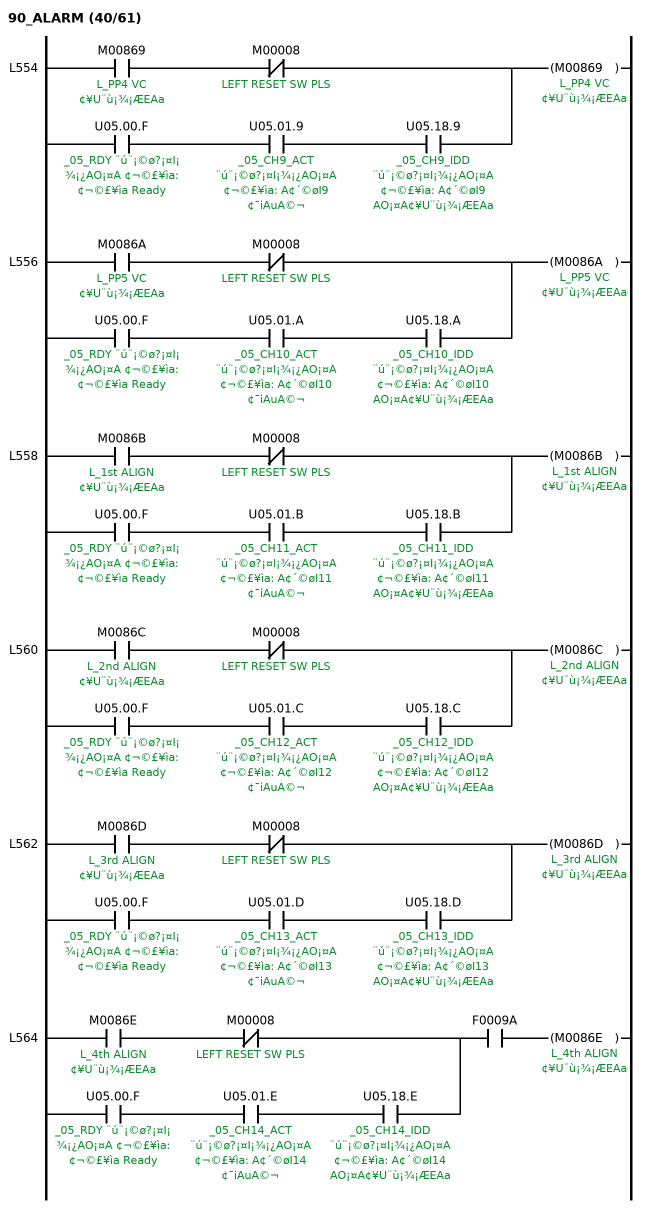
[picture p408: 90_ALARM rungs L554-L564]
; L554
LOAD      M00869	// L_PP4 VC ¢¥U¨ù¡¾¡ÆEAa
AND NOT   M00008	// LEFT RESET SW PLS
LOAD      U05.00.F	// _05_RDY ¨ú¨¡©ø?¡¤I¡¾¡¿AO¡¤A ¢¬©£¥ìa: ¢¬©£¥ìa Ready
AND       U05.01.9	// _05_CH9_ACT ¨ú¨¡©ø?¡¤I¡¾¡¿AO¡¤A ¢¬©£¥ìa: A¢´©øI9 ¢¯iAuA©¬
AND       U05.18.9	// _05_CH9_IDD ¨ú¨¡©ø?¡¤I¡¾¡¿AO¡¤A ¢¬©£¥ìa: A¢´©øI9 AO¡¤A¢¥U¨ù¡¾¡ÆEAa
OR LOAD
OUT       M00869	// L_PP4 VC ¢¥U¨ù¡¾¡ÆEAa
; L556
LOAD      M0086A	// L_PP5 VC ¢¥U¨ù¡¾¡ÆEAa
AND NOT   M00008	// LEFT RESET SW PLS
LOAD      U05.00.F	// _05_RDY ¨ú¨¡©ø?¡¤I¡¾¡¿AO¡¤A ¢¬©£¥ìa: ¢¬©£¥ìa Ready
AND       U05.01.A	// _05_CH10_ACT ¨ú¨¡©ø?¡¤I¡¾¡¿AO¡¤A ¢¬©£¥ìa: A¢´©øI10 ¢¯iAuA©¬
AND       U05.18.A	// _05_CH10_IDD ¨ú¨¡©ø?¡¤I¡¾¡¿AO¡¤A ¢¬©£¥ìa: A¢´©øI10 AO¡¤A¢¥U¨ù¡¾¡ÆEAa
OR LOAD
OUT       M0086A	// L_PP5 VC ¢¥U¨ù¡¾¡ÆEAa
; L558
LOAD      M0086B	// L_1st ALIGN ¢¥U¨ù¡¾¡ÆEAa
AND NOT   M00008	// LEFT RESET SW PLS
LOAD      U05.00.F	// _05_RDY ¨ú¨¡©ø?¡¤I¡¾¡¿AO¡¤A ¢¬©£¥ìa: ¢¬©£¥ìa Ready
AND       U05.01.B	// _05_CH11_ACT ¨ú¨¡©ø?¡¤I¡¾¡¿AO¡¤A ¢¬©£¥ìa: A¢´©øI11 ¢¯iAuA©¬
AND       U05.18.B	// _05_CH11_IDD ¨ú¨¡©ø?¡¤I¡¾¡¿AO¡¤A ¢¬©£¥ìa: A¢´©øI11 AO¡¤A¢¥U¨ù¡¾¡ÆEAa
OR LOAD
OUT       M0086B	// L_1st ALIGN ¢¥U¨ù¡¾¡ÆEAa
; L560
LOAD      M0086C	// L_2nd ALIGN ¢¥U¨ù¡¾¡ÆEAa
AND NOT   M00008	// LEFT RESET SW PLS
LOAD      U05.00.F	// _05_RDY ¨ú¨¡©ø?¡¤I¡¾¡¿AO¡¤A ¢¬©£¥ìa: ¢¬©£¥ìa Ready
AND       U05.01.C	// _05_CH12_ACT ¨ú¨¡©ø?¡¤I¡¾¡¿AO¡¤A ¢¬©£¥ìa: A¢´©øI12 ¢¯iAuA©¬
AND       U05.18.C	// _05_CH12_IDD ¨ú¨¡©ø?¡¤I¡¾¡¿AO¡¤A ¢¬©£¥ìa: A¢´©øI12 AO¡¤A¢¥U¨ù¡¾¡ÆEAa
OR LOAD
OUT       M0086C	// L_2nd ALIGN ¢¥U¨ù¡¾¡ÆEAa
; L562
LOAD      M0086D	// L_3rd ALIGN ¢¥U¨ù¡¾¡ÆEAa
AND NOT   M00008	// LEFT RESET SW PLS
LOAD      U05.00.F	// _05_RDY ¨ú¨¡©ø?¡¤I¡¾¡¿AO¡¤A ¢¬©£¥ìa: ¢¬©£¥ìa Ready
AND       U05.01.D	// _05_CH13_ACT ¨ú¨¡©ø?¡¤I¡¾¡¿AO¡¤A ¢¬©£¥ìa: A¢´©øI13 ¢¯iAuA©¬
AND       U05.18.D	// _05_CH13_IDD ¨ú¨¡©ø?¡¤I¡¾¡¿AO¡¤A ¢¬©£¥ìa: A¢´©øI13 AO¡¤A¢¥U¨ù¡¾¡ÆEAa
OR LOAD
OUT       M0086D	// L_3rd ALIGN ¢¥U¨ù¡¾¡ÆEAa
; L564
LOAD      M0086E	// L_4th ALIGN ¢¥U¨ù¡¾¡ÆEAa
AND NOT   M00008	// LEFT RESET SW PLS
LOAD      U05.00.F	// _05_RDY ¨ú¨¡©ø?¡¤I¡¾¡¿AO¡¤A ¢¬©£¥ìa: ¢¬©£¥ìa Ready
AND       U05.01.E	// _05_CH14_ACT ¨ú¨¡©ø?¡¤I¡¾¡¿AO¡¤A ¢¬©£¥ìa: A¢´©øI14 ¢¯iAuA©¬
AND       U05.18.E	// _05_CH14_IDD ¨ú¨¡©ø?¡¤I¡¾¡¿AO¡¤A ¢¬©£¥ìa: A¢´©øI14 AO¡¤A¢¥U¨ù¡¾¡ÆEAa
OR LOAD
AND       F0009A
OUT       M0086E	// L_4th ALIGN ¢¥U¨ù¡¾¡ÆEAa

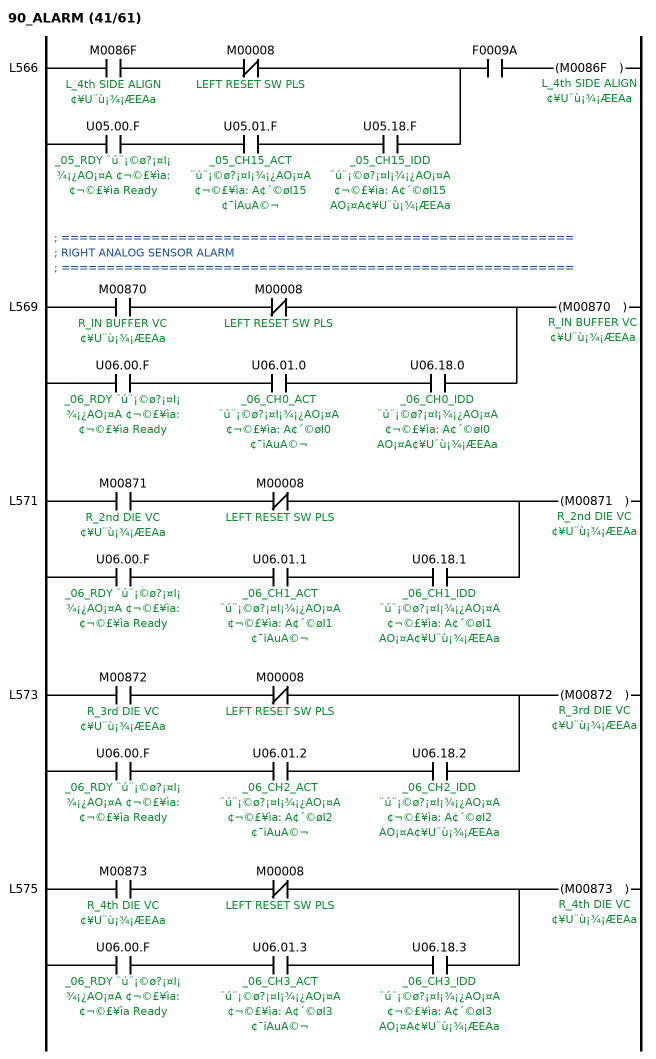
; L566
LOAD      M0086F	// L_4th SIDE ALIGN ¢¥U¨ù¡¾¡ÆEAa
AND NOT   M00008	// LEFT RESET SW PLS
LOAD      U05.00.F	// _05_RDY ¨ú¨¡©ø?¡¤I¡¾¡¿AO¡¤A ¢¬©£¥ìa: ¢¬©£¥ìa Ready
AND       U05.01.F	// _05_CH15_ACT ¨ú¨¡©ø?¡¤I¡¾¡¿AO¡¤A ¢¬©£¥ìa: A¢´©øI15 ¢¯iAuA©¬
AND       U05.18.F	// _05_CH15_IDD ¨ú¨¡©ø?¡¤I¡¾¡¿AO¡¤A ¢¬©£¥ìa: A¢´©øI15 AO¡¤A¢¥U¨ù¡¾¡ÆEAa
OR LOAD
AND       F0009A
OUT       M0086F	// L_4th SIDE ALIGN ¢¥U¨ù¡¾¡ÆEAa
// =========================================================
// 
//        RIGHT ANALOG SENSOR ALARM
// 
// =========================================================
; L569
LOAD      M00870	// R_IN BUFFER VC ¢¥U¨ù¡¾¡ÆEAa
AND NOT   M00008	// LEFT RESET SW PLS
LOAD      U06.00.F	// _06_RDY ¨ú¨¡©ø?¡¤I¡¾¡¿AO¡¤A ¢¬©£¥ìa: ¢¬©£¥ìa Ready
AND       U06.01.0	// _06_CH0_ACT ¨ú¨¡©ø?¡¤I¡¾¡¿AO¡¤A ¢¬©£¥ìa: A¢´©øI0 ¢¯iAuA©¬
AND       U06.18.0	// _06_CH0_IDD ¨ú¨¡©ø?¡¤I¡¾¡¿AO¡¤A ¢¬©£¥ìa: A¢´©øI0 AO¡¤A¢¥U¨ù¡¾¡ÆEAa
OR LOAD
OUT       M00870	// R_IN BUFFER VC ¢¥U¨ù¡¾¡ÆEAa
; L571
LOAD      M00871	// R_2nd DIE VC ¢¥U¨ù¡¾¡ÆEAa
AND NOT   M00008	// LEFT RESET SW PLS
LOAD      U06.00.F	// _06_RDY ¨ú¨¡©ø?¡¤I¡¾¡¿AO¡¤A ¢¬©£¥ìa: ¢¬©£¥ìa Ready
AND       U06.01.1	// _06_CH1_ACT ¨ú¨¡©ø?¡¤I¡¾¡¿AO¡¤A ¢¬©£¥ìa: A¢´©øI1 ¢¯iAuA©¬
AND       U06.18.1	// _06_CH1_IDD ¨ú¨¡©ø?¡¤I¡¾¡¿AO¡¤A ¢¬©£¥ìa: A¢´©øI1 AO¡¤A¢¥U¨ù¡¾¡ÆEAa
OR LOAD
OUT       M00871	// R_2nd DIE VC ¢¥U¨ù¡¾¡ÆEAa
; L573
LOAD      M00872	// R_3rd DIE VC ¢¥U¨ù¡¾¡ÆEAa
AND NOT   M00008	// LEFT RESET SW PLS
LOAD      U06.00.F	// _06_RDY ¨ú¨¡©ø?¡¤I¡¾¡¿AO¡¤A ¢¬©£¥ìa: ¢¬©£¥ìa Ready
AND       U06.01.2	// _06_CH2_ACT ¨ú¨¡©ø?¡¤I¡¾¡¿AO¡¤A ¢¬©£¥ìa: A¢´©øI2 ¢¯iAuA©¬
AND       U06.18.2	// _06_CH2_IDD ¨ú¨¡©ø?¡¤I¡¾¡¿AO¡¤A ¢¬©£¥ìa: A¢´©øI2 AO¡¤A¢¥U¨ù¡¾¡ÆEAa
OR LOAD
OUT       M00872	// R_3rd DIE VC ¢¥U¨ù¡¾¡ÆEAa
; L575
LOAD      M00873	// R_4th DIE VC ¢¥U¨ù¡¾¡ÆEAa
AND NOT   M00008	// LEFT RESET SW PLS
LOAD      U06.00.F	// _06_RDY ¨ú¨¡©ø?¡¤I¡¾¡¿AO¡¤A ¢¬©£¥ìa: ¢¬©£¥ìa Ready
AND       U06.01.3	// _06_CH3_ACT ¨ú¨¡©ø?¡¤I¡¾¡¿AO¡¤A ¢¬©£¥ìa: A¢´©øI3 ¢¯iAuA©¬
AND       U06.18.3	// _06_CH3_IDD ¨ú¨¡©ø?¡¤I¡¾¡¿AO¡¤A ¢¬©£¥ìa: A¢´©øI3 AO¡¤A¢¥U¨ù¡¾¡ÆEAa
OR LOAD
OUT       M00873	// R_4th DIE VC ¢¥U¨ù¡¾¡ÆEAa

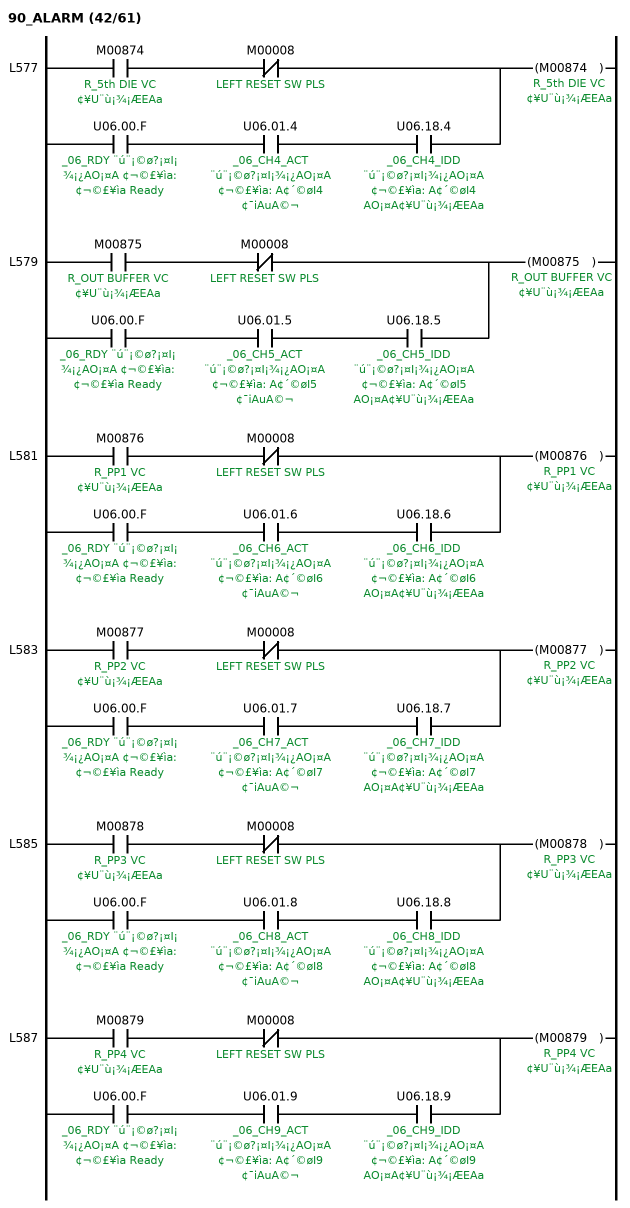
; L577
LOAD      M00874	// R_5th DIE VC ¢¥U¨ù¡¾¡ÆEAa
AND NOT   M00008	// LEFT RESET SW PLS
LOAD      U06.00.F	// _06_RDY ¨ú¨¡©ø?¡¤I¡¾¡¿AO¡¤A ¢¬©£¥ìa: ¢¬©£¥ìa Ready
AND       U06.01.4	// _06_CH4_ACT ¨ú¨¡©ø?¡¤I¡¾¡¿AO¡¤A ¢¬©£¥ìa: A¢´©øI4 ¢¯iAuA©¬
AND       U06.18.4	// _06_CH4_IDD ¨ú¨¡©ø?¡¤I¡¾¡¿AO¡¤A ¢¬©£¥ìa: A¢´©øI4 AO¡¤A¢¥U¨ù¡¾¡ÆEAa
OR LOAD
OUT       M00874	// R_5th DIE VC ¢¥U¨ù¡¾¡ÆEAa
; L579
LOAD      M00875	// R_OUT BUFFER VC ¢¥U¨ù¡¾¡ÆEAa
AND NOT   M00008	// LEFT RESET SW PLS
LOAD      U06.00.F	// _06_RDY ¨ú¨¡©ø?¡¤I¡¾¡¿AO¡¤A ¢¬©£¥ìa: ¢¬©£¥ìa Ready
AND       U06.01.5	// _06_CH5_ACT ¨ú¨¡©ø?¡¤I¡¾¡¿AO¡¤A ¢¬©£¥ìa: A¢´©øI5 ¢¯iAuA©¬
AND       U06.18.5	// _06_CH5_IDD ¨ú¨¡©ø?¡¤I¡¾¡¿AO¡¤A ¢¬©£¥ìa: A¢´©øI5 AO¡¤A¢¥U¨ù¡¾¡ÆEAa
OR LOAD
OUT       M00875	// R_OUT BUFFER VC ¢¥U¨ù¡¾¡ÆEAa
; L581
LOAD      M00876	// R_PP1 VC ¢¥U¨ù¡¾¡ÆEAa
AND NOT   M00008	// LEFT RESET SW PLS
LOAD      U06.00.F	// _06_RDY ¨ú¨¡©ø?¡¤I¡¾¡¿AO¡¤A ¢¬©£¥ìa: ¢¬©£¥ìa Ready
AND       U06.01.6	// _06_CH6_ACT ¨ú¨¡©ø?¡¤I¡¾¡¿AO¡¤A ¢¬©£¥ìa: A¢´©øI6 ¢¯iAuA©¬
AND       U06.18.6	// _06_CH6_IDD ¨ú¨¡©ø?¡¤I¡¾¡¿AO¡¤A ¢¬©£¥ìa: A¢´©øI6 AO¡¤A¢¥U¨ù¡¾¡ÆEAa
OR LOAD
OUT       M00876	// R_PP1 VC ¢¥U¨ù¡¾¡ÆEAa
; L583
LOAD      M00877	// R_PP2 VC ¢¥U¨ù¡¾¡ÆEAa
AND NOT   M00008	// LEFT RESET SW PLS
LOAD      U06.00.F	// _06_RDY ¨ú¨¡©ø?¡¤I¡¾¡¿AO¡¤A ¢¬©£¥ìa: ¢¬©£¥ìa Ready
AND       U06.01.7	// _06_CH7_ACT ¨ú¨¡©ø?¡¤I¡¾¡¿AO¡¤A ¢¬©£¥ìa: A¢´©øI7 ¢¯iAuA©¬
AND       U06.18.7	// _06_CH7_IDD ¨ú¨¡©ø?¡¤I¡¾¡¿AO¡¤A ¢¬©£¥ìa: A¢´©øI7 AO¡¤A¢¥U¨ù¡¾¡ÆEAa
OR LOAD
OUT       M00877	// R_PP2 VC ¢¥U¨ù¡¾¡ÆEAa
; L585
LOAD      M00878	// R_PP3 VC ¢¥U¨ù¡¾¡ÆEAa
AND NOT   M00008	// LEFT RESET SW PLS
LOAD      U06.00.F	// _06_RDY ¨ú¨¡©ø?¡¤I¡¾¡¿AO¡¤A ¢¬©£¥ìa: ¢¬©£¥ìa Ready
AND       U06.01.8	// _06_CH8_ACT ¨ú¨¡©ø?¡¤I¡¾¡¿AO¡¤A ¢¬©£¥ìa: A¢´©øI8 ¢¯iAuA©¬
AND       U06.18.8	// _06_CH8_IDD ¨ú¨¡©ø?¡¤I¡¾¡¿AO¡¤A ¢¬©£¥ìa: A¢´©øI8 AO¡¤A¢¥U¨ù¡¾¡ÆEAa
OR LOAD
OUT       M00878	// R_PP3 VC ¢¥U¨ù¡¾¡ÆEAa
; L587
LOAD      M00879	// R_PP4 VC ¢¥U¨ù¡¾¡ÆEAa
AND NOT   M00008	// LEFT RESET SW PLS
LOAD      U06.00.F	// _06_RDY ¨ú¨¡©ø?¡¤I¡¾¡¿AO¡¤A ¢¬©£¥ìa: ¢¬©£¥ìa Ready
AND       U06.01.9	// _06_CH9_ACT ¨ú¨¡©ø?¡¤I¡¾¡¿AO¡¤A ¢¬©£¥ìa: A¢´©øI9 ¢¯iAuA©¬
AND       U06.18.9	// _06_CH9_IDD ¨ú¨¡©ø?¡¤I¡¾¡¿AO¡¤A ¢¬©£¥ìa: A¢´©øI9 AO¡¤A¢¥U¨ù¡¾¡ÆEAa
OR LOAD
OUT       M00879	// R_PP4 VC ¢¥U¨ù¡¾¡ÆEAa

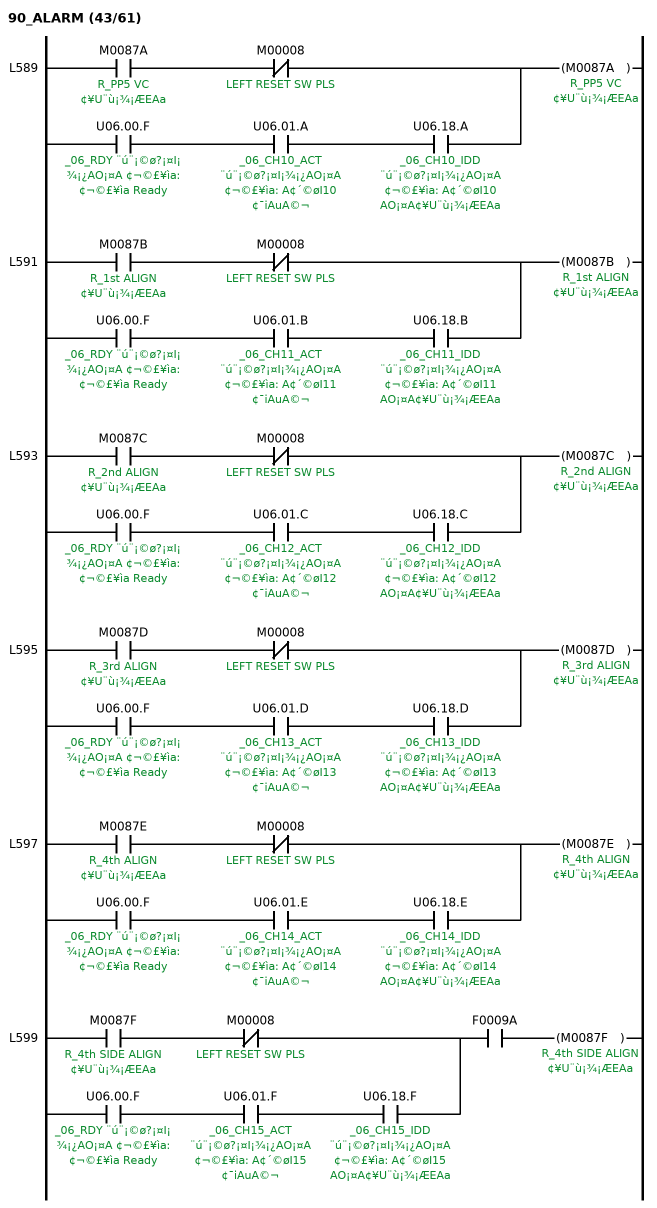
; L589
LOAD      M0087A	// R_PP5 VC ¢¥U¨ù¡¾¡ÆEAa
AND NOT   M00008	// LEFT RESET SW PLS
LOAD      U06.00.F	// _06_RDY ¨ú¨¡©ø?¡¤I¡¾¡¿AO¡¤A ¢¬©£¥ìa: ¢¬©£¥ìa Ready
AND       U06.01.A	// _06_CH10_ACT ¨ú¨¡©ø?¡¤I¡¾¡¿AO¡¤A ¢¬©£¥ìa: A¢´©øI10 ¢¯iAuA©¬
AND       U06.18.A	// _06_CH10_IDD ¨ú¨¡©ø?¡¤I¡¾¡¿AO¡¤A ¢¬©£¥ìa: A¢´©øI10 AO¡¤A¢¥U¨ù¡¾¡ÆEAa
OR LOAD
OUT       M0087A	// R_PP5 VC ¢¥U¨ù¡¾¡ÆEAa
; L591
LOAD      M0087B	// R_1st ALIGN ¢¥U¨ù¡¾¡ÆEAa
AND NOT   M00008	// LEFT RESET SW PLS
LOAD      U06.00.F	// _06_RDY ¨ú¨¡©ø?¡¤I¡¾¡¿AO¡¤A ¢¬©£¥ìa: ¢¬©£¥ìa Ready
AND       U06.01.B	// _06_CH11_ACT ¨ú¨¡©ø?¡¤I¡¾¡¿AO¡¤A ¢¬©£¥ìa: A¢´©øI11 ¢¯iAuA©¬
AND       U06.18.B	// _06_CH11_IDD ¨ú¨¡©ø?¡¤I¡¾¡¿AO¡¤A ¢¬©£¥ìa: A¢´©øI11 AO¡¤A¢¥U¨ù¡¾¡ÆEAa
OR LOAD
OUT       M0087B	// R_1st ALIGN ¢¥U¨ù¡¾¡ÆEAa
; L593
LOAD      M0087C	// R_2nd ALIGN ¢¥U¨ù¡¾¡ÆEAa
AND NOT   M00008	// LEFT RESET SW PLS
LOAD      U06.00.F	// _06_RDY ¨ú¨¡©ø?¡¤I¡¾¡¿AO¡¤A ¢¬©£¥ìa: ¢¬©£¥ìa Ready
AND       U06.01.C	// _06_CH12_ACT ¨ú¨¡©ø?¡¤I¡¾¡¿AO¡¤A ¢¬©£¥ìa: A¢´©øI12 ¢¯iAuA©¬
AND       U06.18.C	// _06_CH12_IDD ¨ú¨¡©ø?¡¤I¡¾¡¿AO¡¤A ¢¬©£¥ìa: A¢´©øI12 AO¡¤A¢¥U¨ù¡¾¡ÆEAa
OR LOAD
OUT       M0087C	// R_2nd ALIGN ¢¥U¨ù¡¾¡ÆEAa
; L595
LOAD      M0087D	// R_3rd ALIGN ¢¥U¨ù¡¾¡ÆEAa
AND NOT   M00008	// LEFT RESET SW PLS
LOAD      U06.00.F	// _06_RDY ¨ú¨¡©ø?¡¤I¡¾¡¿AO¡¤A ¢¬©£¥ìa: ¢¬©£¥ìa Ready
AND       U06.01.D	// _06_CH13_ACT ¨ú¨¡©ø?¡¤I¡¾¡¿AO¡¤A ¢¬©£¥ìa: A¢´©øI13 ¢¯iAuA©¬
AND       U06.18.D	// _06_CH13_IDD ¨ú¨¡©ø?¡¤I¡¾¡¿AO¡¤A ¢¬©£¥ìa: A¢´©øI13 AO¡¤A¢¥U¨ù¡¾¡ÆEAa
OR LOAD
OUT       M0087D	// R_3rd ALIGN ¢¥U¨ù¡¾¡ÆEAa
; L597
LOAD      M0087E	// R_4th ALIGN ¢¥U¨ù¡¾¡ÆEAa
AND NOT   M00008	// LEFT RESET SW PLS
LOAD      U06.00.F	// _06_RDY ¨ú¨¡©ø?¡¤I¡¾¡¿AO¡¤A ¢¬©£¥ìa: ¢¬©£¥ìa Ready
AND       U06.01.E	// _06_CH14_ACT ¨ú¨¡©ø?¡¤I¡¾¡¿AO¡¤A ¢¬©£¥ìa: A¢´©øI14 ¢¯iAuA©¬
AND       U06.18.E	// _06_CH14_IDD ¨ú¨¡©ø?¡¤I¡¾¡¿AO¡¤A ¢¬©£¥ìa: A¢´©øI14 AO¡¤A¢¥U¨ù¡¾¡ÆEAa
OR LOAD
OUT       M0087E	// R_4th ALIGN ¢¥U¨ù¡¾¡ÆEAa
; L599
LOAD      M0087F	// R_4th SIDE ALIGN ¢¥U¨ù¡¾¡ÆEAa
AND NOT   M00008	// LEFT RESET SW PLS
LOAD      U06.00.F	// _06_RDY ¨ú¨¡©ø?¡¤I¡¾¡¿AO¡¤A ¢¬©£¥ìa: ¢¬©£¥ìa Ready
AND       U06.01.F	// _06_CH15_ACT ¨ú¨¡©ø?¡¤I¡¾¡¿AO¡¤A ¢¬©£¥ìa: A¢´©øI15 ¢¯iAuA©¬
AND       U06.18.F	// _06_CH15_IDD ¨ú¨¡©ø?¡¤I¡¾¡¿AO¡¤A ¢¬©£¥ìa: A¢´©øI15 AO¡¤A¢¥U¨ù¡¾¡ÆEAa
OR LOAD
AND       F0009A
OUT       M0087F	// R_4th SIDE ALIGN ¢¥U¨ù¡¾¡ÆEAa

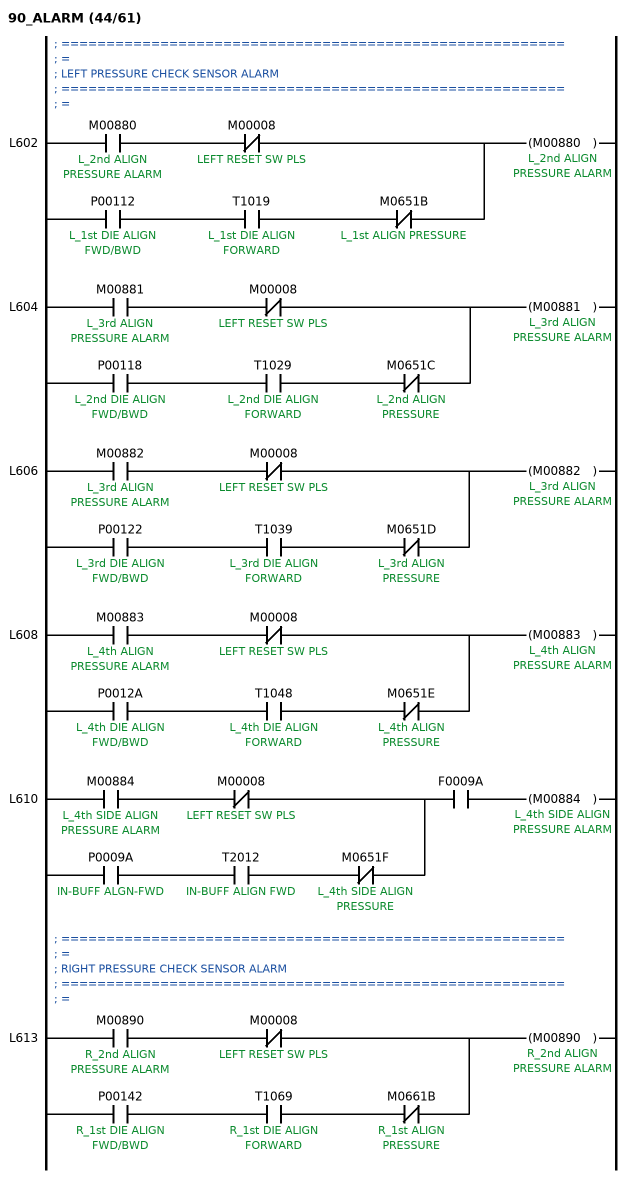
// =========================================================
// 
//        LEFT PRESSURE CHECK SENSOR ALARM
// 
// =========================================================
; L602
LOAD      M00880	// L_2nd ALIGN PRESSURE ALARM
AND NOT   M00008	// LEFT RESET SW PLS
LOAD      P00112	// L_1st DIE ALIGN FWD/BWD
AND       T1019	// L_1st DIE ALIGN FORWARD
AND NOT   M0651B	// L_1st ALIGN PRESSURE
OR LOAD
OUT       M00880	// L_2nd ALIGN PRESSURE ALARM
; L604
LOAD      M00881	// L_3rd ALIGN PRESSURE ALARM
AND NOT   M00008	// LEFT RESET SW PLS
LOAD      P00118	// L_2nd DIE ALIGN FWD/BWD
AND       T1029	// L_2nd DIE ALIGN FORWARD
AND NOT   M0651C	// L_2nd ALIGN PRESSURE
OR LOAD
OUT       M00881	// L_3rd ALIGN PRESSURE ALARM
; L606
LOAD      M00882	// L_3rd ALIGN PRESSURE ALARM
AND NOT   M00008	// LEFT RESET SW PLS
LOAD      P00122	// L_3rd DIE ALIGN FWD/BWD
AND       T1039	// L_3rd DIE ALIGN FORWARD
AND NOT   M0651D	// L_3rd ALIGN PRESSURE
OR LOAD
OUT       M00882	// L_3rd ALIGN PRESSURE ALARM
; L608
LOAD      M00883	// L_4th ALIGN PRESSURE ALARM
AND NOT   M00008	// LEFT RESET SW PLS
LOAD      P0012A	// L_4th DIE ALIGN FWD/BWD
AND       T1048	// L_4th DIE ALIGN FORWARD
AND NOT   M0651E	// L_4th ALIGN PRESSURE
OR LOAD
OUT       M00883	// L_4th ALIGN PRESSURE ALARM
; L610
LOAD      M00884	// L_4th SIDE ALIGN PRESSURE ALARM
AND NOT   M00008	// LEFT RESET SW PLS
LOAD      P0009A	// IN-BUFF ALGN-FWD
AND       T2012	// IN-BUFF ALIGN FWD
AND NOT   M0651F	// L_4th SIDE ALIGN PRESSURE
OR LOAD
AND       F0009A
OUT       M00884	// L_4th SIDE ALIGN PRESSURE ALARM
// =========================================================
// 
//        RIGHT PRESSURE CHECK SENSOR ALARM
// 
// =========================================================
; L613
LOAD      M00890	// R_2nd ALIGN PRESSURE ALARM
AND NOT   M00008	// LEFT RESET SW PLS
LOAD      P00142	// R_1st DIE ALIGN FWD/BWD
AND       T1069	// R_1st DIE ALIGN FORWARD
AND NOT   M0661B	// R_1st ALIGN PRESSURE
OR LOAD
OUT       M00890	// R_2nd ALIGN PRESSURE ALARM

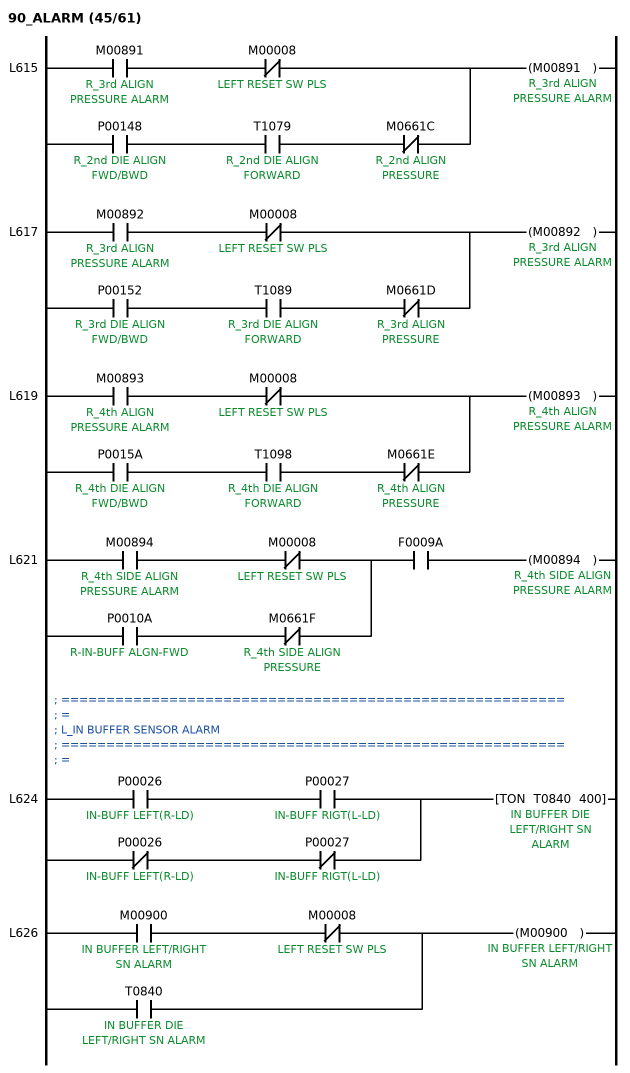
; L615
LOAD      M00891	// R_3rd ALIGN PRESSURE ALARM
AND NOT   M00008	// LEFT RESET SW PLS
LOAD      P00148	// R_2nd DIE ALIGN FWD/BWD
AND       T1079	// R_2nd DIE ALIGN FORWARD
AND NOT   M0661C	// R_2nd ALIGN PRESSURE
OR LOAD
OUT       M00891	// R_3rd ALIGN PRESSURE ALARM
; L617
LOAD      M00892	// R_3rd ALIGN PRESSURE ALARM
AND NOT   M00008	// LEFT RESET SW PLS
LOAD      P00152	// R_3rd DIE ALIGN FWD/BWD
AND       T1089	// R_3rd DIE ALIGN FORWARD
AND NOT   M0661D	// R_3rd ALIGN PRESSURE
OR LOAD
OUT       M00892	// R_3rd ALIGN PRESSURE ALARM
; L619
LOAD      M00893	// R_4th ALIGN PRESSURE ALARM
AND NOT   M00008	// LEFT RESET SW PLS
LOAD      P0015A	// R_4th DIE ALIGN FWD/BWD
AND       T1098	// R_4th DIE ALIGN FORWARD
AND NOT   M0661E	// R_4th ALIGN PRESSURE
OR LOAD
OUT       M00893	// R_4th ALIGN PRESSURE ALARM
; L621
LOAD      M00894	// R_4th SIDE ALIGN PRESSURE ALARM
AND NOT   M00008	// LEFT RESET SW PLS
LOAD      P0010A	// R-IN-BUFF ALGN-FWD
AND NOT   M0661F	// R_4th SIDE ALIGN PRESSURE
OR LOAD
AND       F0009A
OUT       M00894	// R_4th SIDE ALIGN PRESSURE ALARM
// =========================================================
// 
//        L_IN BUFFER SENSOR ALARM
// 
// =========================================================
; L624
LOAD      P00026	// IN-BUFF LEFT(R-LD)
AND       P00027	// IN-BUFF RIGT(L-LD)
LOAD NOT  P00026	// IN-BUFF LEFT(R-LD)
AND NOT   P00027	// IN-BUFF RIGT(L-LD)
OR LOAD
TON       T0840 400	// IN BUFFER DIE LEFT/RIGHT SN ALARM
; L626
LOAD      M00900	// IN BUFFER LEFT/RIGHT SN ALARM
AND NOT   M00008	// LEFT RESET SW PLS
OR        T0840	// IN BUFFER DIE LEFT/RIGHT SN ALARM
OUT       M00900	// IN BUFFER LEFT/RIGHT SN ALARM

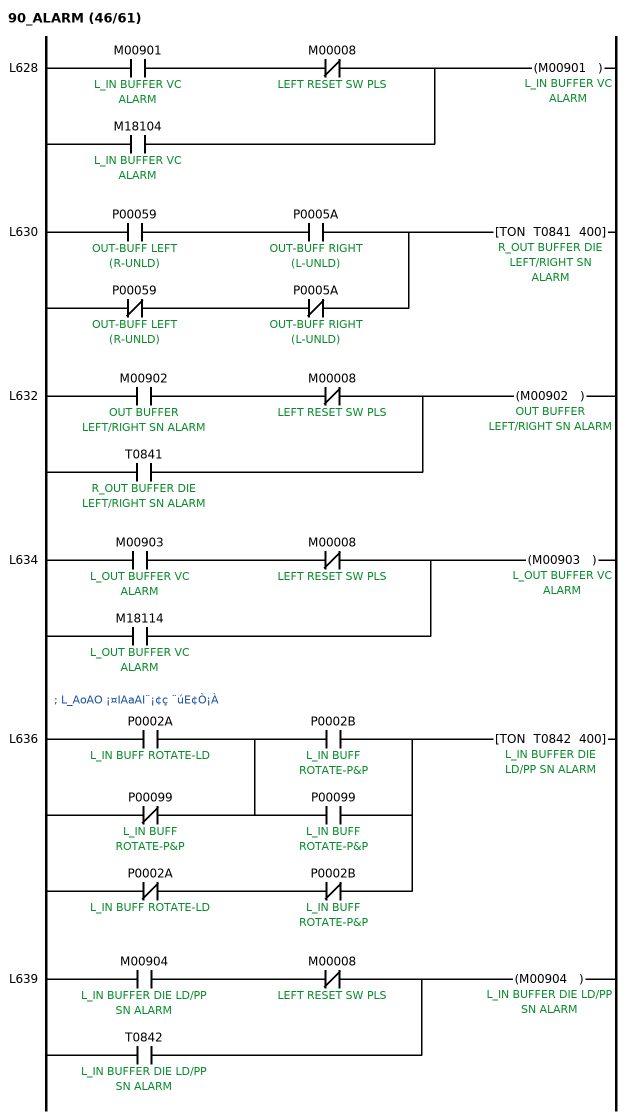
; L628
LOAD      M00901	// L_IN BUFFER VC ALARM
AND NOT   M00008	// LEFT RESET SW PLS
OR        M18104	// L_IN BUFFER VC ALARM
OUT       M00901	// L_IN BUFFER VC ALARM
; L630
LOAD      P00059	// OUT-BUFF LEFT (R-UNLD)
AND       P0005A	// OUT-BUFF RIGHT (L-UNLD)
LOAD NOT  P00059	// OUT-BUFF LEFT (R-UNLD)
AND NOT   P0005A	// OUT-BUFF RIGHT (L-UNLD)
OR LOAD
TON       T0841 400	// R_OUT BUFFER DIE LEFT/RIGHT SN ALARM
; L632
LOAD      M00902	// OUT BUFFER LEFT/RIGHT SN ALARM
AND NOT   M00008	// LEFT RESET SW PLS
OR        T0841	// R_OUT BUFFER DIE LEFT/RIGHT SN ALARM
OUT       M00902	// OUT BUFFER LEFT/RIGHT SN ALARM
; L634
LOAD      M00903	// L_OUT BUFFER VC ALARM
AND NOT   M00008	// LEFT RESET SW PLS
OR        M18114	// L_OUT BUFFER VC ALARM
OUT       M00903	// L_OUT BUFFER VC ALARM
; L636
LOAD      P0002A	// L_IN BUFF ROTATE-LD
OR NOT    P00099	// L_IN BUFF ROTATE-P&P
LOAD      P0002B	// L_IN BUFF ROTATE-P&P
OR        P00099	// L_IN BUFF ROTATE-P&P
AND LOAD
LOAD NOT  P0002A	// L_IN BUFF ROTATE-LD
AND NOT   P0002B	// L_IN BUFF ROTATE-P&P
OR LOAD
TON       T0842 400	// L_IN BUFFER DIE LD/PP SN ALARM
// output comment: L_AoAO ¡¤IAaAI¨¡¢ç ¨úE¢Ò¡À
; L639
LOAD      M00904	// L_IN BUFFER DIE LD/PP SN ALARM
AND NOT   M00008	// LEFT RESET SW PLS
OR        T0842	// L_IN BUFFER DIE LD/PP SN ALARM
OUT       M00904	// L_IN BUFFER DIE LD/PP SN ALARM

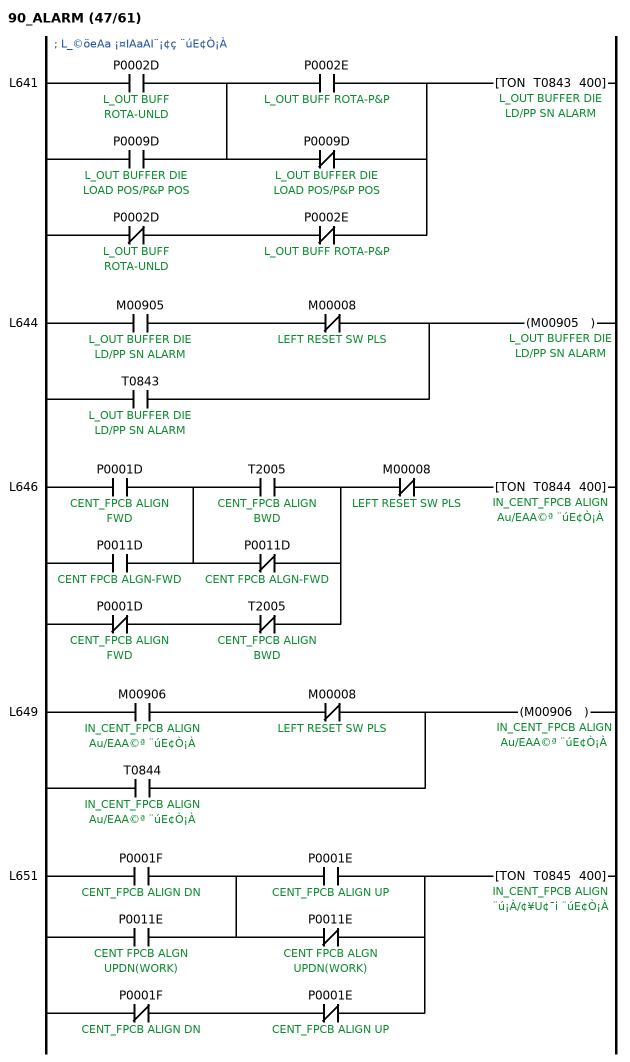
; L641
LOAD      P0002D	// L_OUT BUFF ROTA-UNLD
OR        P0009D	// L_OUT BUFFER DIE LOAD POS/P&P POS
LOAD      P0002E	// L_OUT BUFF ROTA-P&P
OR NOT    P0009D	// L_OUT BUFFER DIE LOAD POS/P&P POS
AND LOAD
LOAD NOT  P0002D	// L_OUT BUFF ROTA-UNLD
AND NOT   P0002E	// L_OUT BUFF ROTA-P&P
OR LOAD
TON       T0843 400	// L_OUT BUFFER DIE LD/PP SN ALARM
// output comment: L_©öeAa ¡¤IAaAI¨¡¢ç ¨úE¢Ò¡À
; L644
LOAD      M00905	// L_OUT BUFFER DIE LD/PP SN ALARM
AND NOT   M00008	// LEFT RESET SW PLS
OR        T0843	// L_OUT BUFFER DIE LD/PP SN ALARM
OUT       M00905	// L_OUT BUFFER DIE LD/PP SN ALARM
; L646
LOAD      P0001D	// CENT_FPCB ALIGN FWD
OR        P0011D	// CENT FPCB ALGN-FWD
LOAD      T2005	// CENT_FPCB ALIGN BWD
OR NOT    P0011D	// CENT FPCB ALGN-FWD
AND LOAD
LOAD NOT  P0001D	// CENT_FPCB ALIGN FWD
AND NOT   T2005	// CENT_FPCB ALIGN BWD
OR LOAD
AND NOT   M00008	// LEFT RESET SW PLS
TON       T0844 400	// IN_CENT_FPCB ALIGN Au/EAA©ª ¨úE¢Ò¡À
; L649
LOAD      M00906	// IN_CENT_FPCB ALIGN Au/EAA©ª ¨úE¢Ò¡À
AND NOT   M00008	// LEFT RESET SW PLS
OR        T0844	// IN_CENT_FPCB ALIGN Au/EAA©ª ¨úE¢Ò¡À
OUT       M00906	// IN_CENT_FPCB ALIGN Au/EAA©ª ¨úE¢Ò¡À
; L651
LOAD      P0001F	// CENT_FPCB ALIGN DN
OR        P0011E	// CENT FPCB ALGN UPDN(WORK)
LOAD      P0001E	// CENT_FPCB ALIGN UP
OR NOT    P0011E	// CENT FPCB ALGN UPDN(WORK)
AND LOAD
LOAD NOT  P0001F	// CENT_FPCB ALIGN DN
AND NOT   P0001E	// CENT_FPCB ALIGN UP
OR LOAD
TON       T0845 400	// IN_CENT_FPCB ALIGN ¨ú¡À/¢¥U¢¯i ¨úE¢Ò¡À

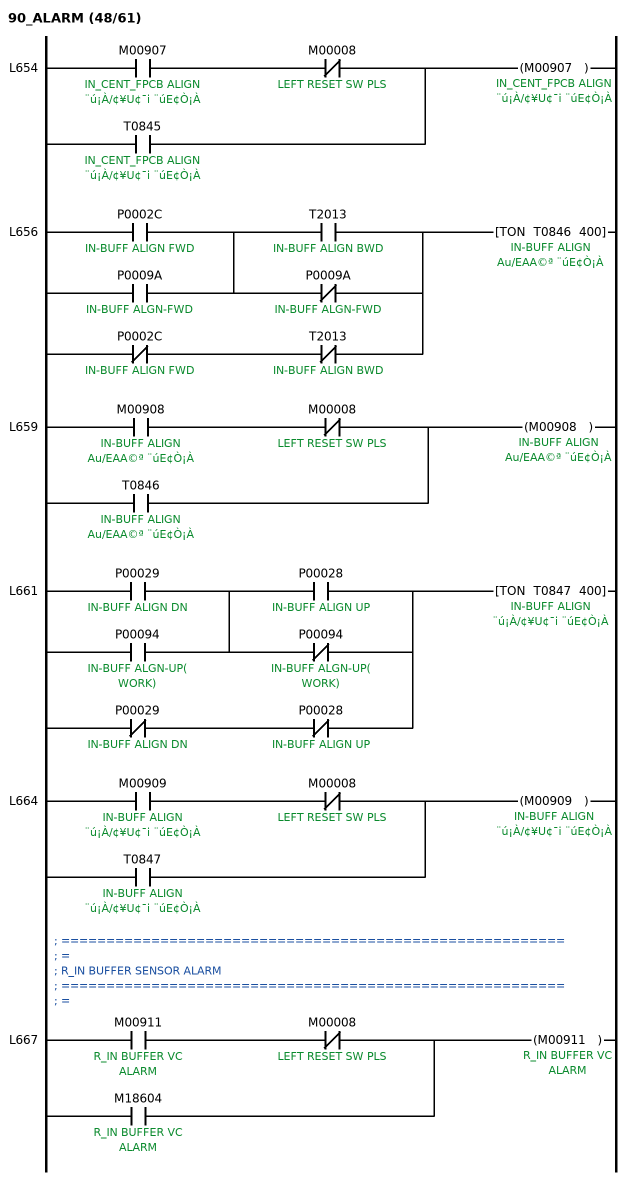
; L654
LOAD      M00907	// IN_CENT_FPCB ALIGN ¨ú¡À/¢¥U¢¯i ¨úE¢Ò¡À
AND NOT   M00008	// LEFT RESET SW PLS
OR        T0845	// IN_CENT_FPCB ALIGN ¨ú¡À/¢¥U¢¯i ¨úE¢Ò¡À
OUT       M00907	// IN_CENT_FPCB ALIGN ¨ú¡À/¢¥U¢¯i ¨úE¢Ò¡À
; L656
LOAD      P0002C	// IN-BUFF ALIGN FWD
OR        P0009A	// IN-BUFF ALGN-FWD
LOAD      T2013	// IN-BUFF ALIGN BWD
OR NOT    P0009A	// IN-BUFF ALGN-FWD
AND LOAD
LOAD NOT  P0002C	// IN-BUFF ALIGN FWD
AND NOT   T2013	// IN-BUFF ALIGN BWD
OR LOAD
TON       T0846 400	// IN-BUFF ALIGN Au/EAA©ª ¨úE¢Ò¡À
; L659
LOAD      M00908	// IN-BUFF ALIGN Au/EAA©ª ¨úE¢Ò¡À
AND NOT   M00008	// LEFT RESET SW PLS
OR        T0846	// IN-BUFF ALIGN Au/EAA©ª ¨úE¢Ò¡À
OUT       M00908	// IN-BUFF ALIGN Au/EAA©ª ¨úE¢Ò¡À
; L661
LOAD      P00029	// IN-BUFF ALIGN DN
OR        P00094	// IN-BUFF ALGN-UP(WORK)
LOAD      P00028	// IN-BUFF ALIGN UP
OR NOT    P00094	// IN-BUFF ALGN-UP(WORK)
AND LOAD
LOAD NOT  P00029	// IN-BUFF ALIGN DN
AND NOT   P00028	// IN-BUFF ALIGN UP
OR LOAD
TON       T0847 400	// IN-BUFF ALIGN ¨ú¡À/¢¥U¢¯i ¨úE¢Ò¡À
; L664
LOAD      M00909	// IN-BUFF ALIGN ¨ú¡À/¢¥U¢¯i ¨úE¢Ò¡À
AND NOT   M00008	// LEFT RESET SW PLS
OR        T0847	// IN-BUFF ALIGN ¨ú¡À/¢¥U¢¯i ¨úE¢Ò¡À
OUT       M00909	// IN-BUFF ALIGN ¨ú¡À/¢¥U¢¯i ¨úE¢Ò¡À
// =========================================================
// 
//        R_IN BUFFER SENSOR ALARM
// 
// =========================================================
; L667
LOAD      M00911	// R_IN BUFFER VC ALARM
AND NOT   M00008	// LEFT RESET SW PLS
OR        M18604	// R_IN BUFFER VC ALARM
OUT       M00911	// R_IN BUFFER VC ALARM

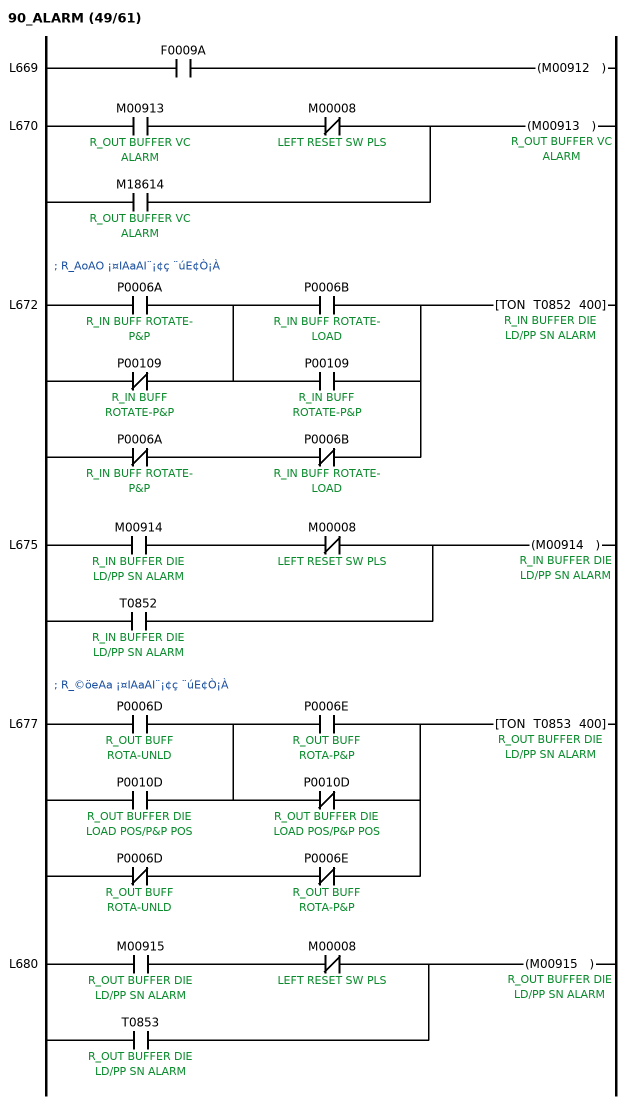
; L669
LOAD      F0009A
OUT       M00912
; L670
LOAD      M00913	// R_OUT BUFFER VC ALARM
AND NOT   M00008	// LEFT RESET SW PLS
OR        M18614	// R_OUT BUFFER VC ALARM
OUT       M00913	// R_OUT BUFFER VC ALARM
; L672
LOAD      P0006A	// R_IN BUFF ROTATE- P&P
OR NOT    P00109	// R_IN BUFF ROTATE-P&P
LOAD      P0006B	// R_IN BUFF ROTATE- LOAD
OR        P00109	// R_IN BUFF ROTATE-P&P
AND LOAD
LOAD NOT  P0006A	// R_IN BUFF ROTATE- P&P
AND NOT   P0006B	// R_IN BUFF ROTATE- LOAD
OR LOAD
TON       T0852 400	// R_IN BUFFER DIE LD/PP SN ALARM
// output comment: R_AoAO ¡¤IAaAI¨¡¢ç ¨úE¢Ò¡À
; L675
LOAD      M00914	// R_IN BUFFER DIE LD/PP SN ALARM
AND NOT   M00008	// LEFT RESET SW PLS
OR        T0852	// R_IN BUFFER DIE LD/PP SN ALARM
OUT       M00914	// R_IN BUFFER DIE LD/PP SN ALARM
; L677
LOAD      P0006D	// R_OUT BUFF ROTA-UNLD
OR        P0010D	// R_OUT BUFFER DIE LOAD POS/P&P POS
LOAD      P0006E	// R_OUT BUFF ROTA-P&P
OR NOT    P0010D	// R_OUT BUFFER DIE LOAD POS/P&P POS
AND LOAD
LOAD NOT  P0006D	// R_OUT BUFF ROTA-UNLD
AND NOT   P0006E	// R_OUT BUFF ROTA-P&P
OR LOAD
TON       T0853 400	// R_OUT BUFFER DIE LD/PP SN ALARM
// output comment: R_©öeAa ¡¤IAaAI¨¡¢ç ¨úE¢Ò¡À
; L680
LOAD      M00915	// R_OUT BUFFER DIE LD/PP SN ALARM
AND NOT   M00008	// LEFT RESET SW PLS
OR        T0853	// R_OUT BUFFER DIE LD/PP SN ALARM
OUT       M00915	// R_OUT BUFFER DIE LD/PP SN ALARM

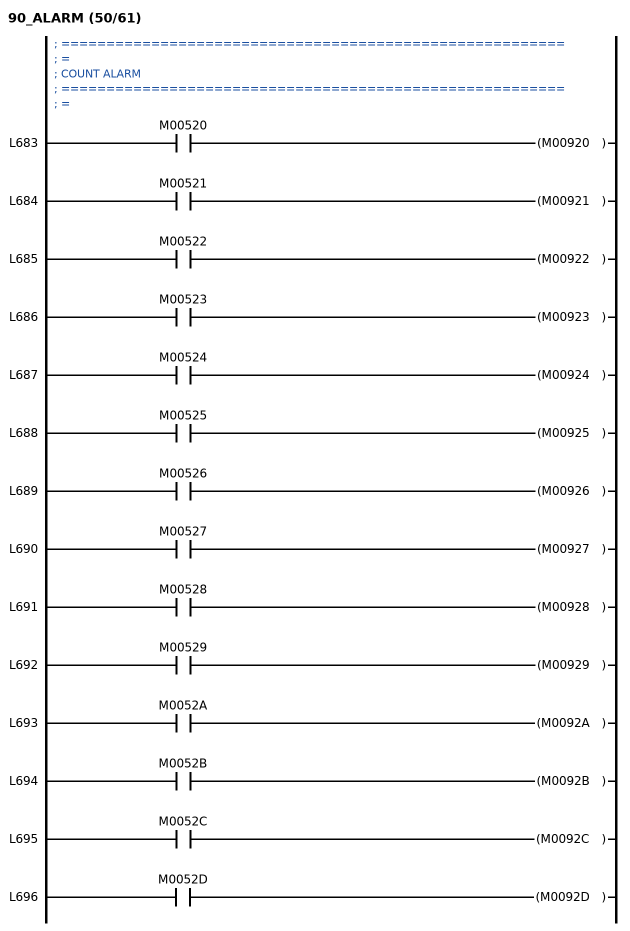
// =========================================================
// 
//       COUNT ALARM
// 
// =========================================================
; L683
LOAD      M00520
OUT       M00920
; L684
LOAD      M00521
OUT       M00921
; L685
LOAD      M00522
OUT       M00922
; L686
LOAD      M00523
OUT       M00923
; L687
LOAD      M00524
OUT       M00924
; L688
LOAD      M00525
OUT       M00925
; L689
LOAD      M00526
OUT       M00926
; L690
LOAD      M00527
OUT       M00927
; L691
LOAD      M00528
OUT       M00928
; L692
LOAD      M00529
OUT       M00929
; L693
LOAD      M0052A
OUT       M0092A
; L694
LOAD      M0052B
OUT       M0092B
; L695
LOAD      M0052C
OUT       M0092C
; L696
LOAD      M0052D
OUT       M0092D

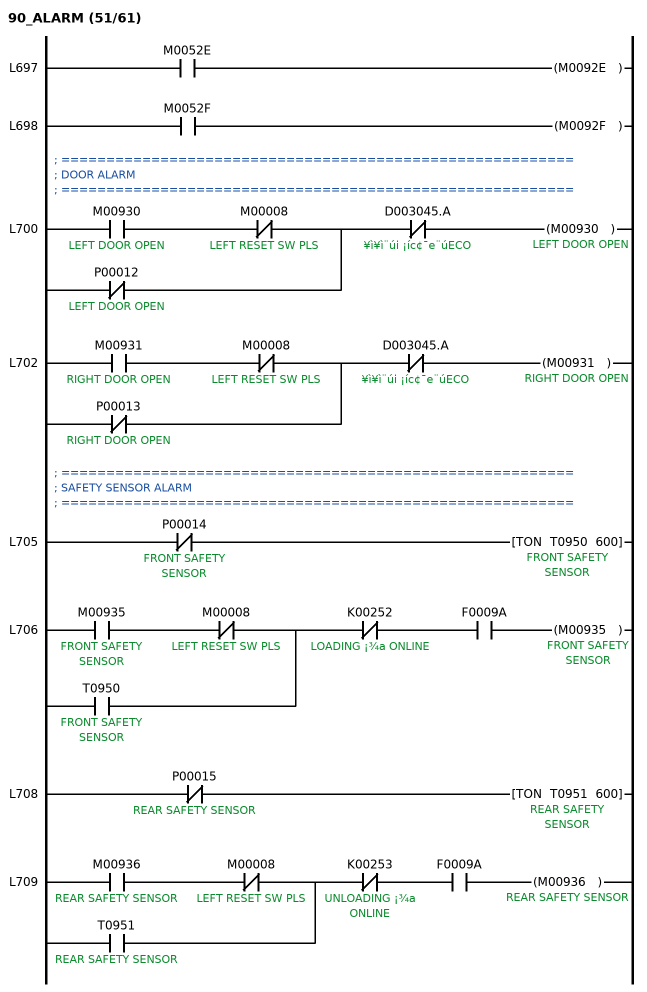
; L697
LOAD      M0052E
OUT       M0092E
; L698
LOAD      M0052F
OUT       M0092F
// =========================================================
// 
//       DOOR ALARM
// 
// =========================================================
; L700
LOAD      M00930	// LEFT DOOR OPEN
AND NOT   M00008	// LEFT RESET SW PLS
OR NOT    P00012	// LEFT DOOR OPEN
AND NOT   D003045.A	// ¥ì¥ì¨úi ¡íc¢¯e¨úECO
OUT       M00930	// LEFT DOOR OPEN
; L702
LOAD      M00931	// RIGHT DOOR OPEN
AND NOT   M00008	// LEFT RESET SW PLS
OR NOT    P00013	// RIGHT DOOR OPEN
AND NOT   D003045.A	// ¥ì¥ì¨úi ¡íc¢¯e¨úECO
OUT       M00931	// RIGHT DOOR OPEN
// =========================================================
// 
//       SAFETY SENSOR ALARM
// 
// =========================================================
; L705
LOAD NOT  P00014	// FRONT SAFETY SENSOR
TON       T0950 600	// FRONT SAFETY SENSOR
; L706
LOAD      M00935	// FRONT SAFETY SENSOR
AND NOT   M00008	// LEFT RESET SW PLS
OR        T0950	// FRONT SAFETY SENSOR
AND NOT   K00252	// LOADING ¡¾a ONLINE
AND       F0009A
OUT       M00935	// FRONT SAFETY SENSOR
; L708
LOAD NOT  P00015	// REAR SAFETY SENSOR
TON       T0951 600	// REAR SAFETY SENSOR
; L709
LOAD      M00936	// REAR SAFETY SENSOR
AND NOT   M00008	// LEFT RESET SW PLS
OR        T0951	// REAR SAFETY SENSOR
AND NOT   K00253	// UNLOADING ¡¾a ONLINE
AND       F0009A
OUT       M00936	// REAR SAFETY SENSOR

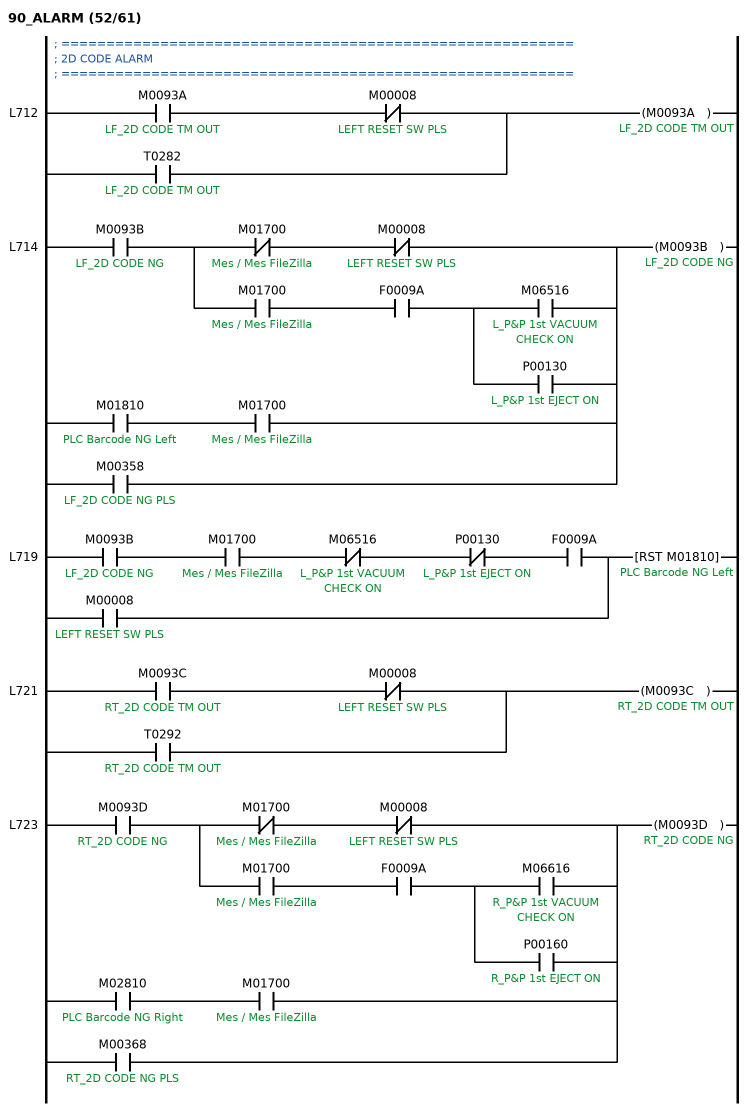
// =========================================================
// 
//       2D CODE ALARM
// 
// =========================================================
; L712
LOAD      M0093A	// LF_2D CODE TM OUT
AND NOT   M00008	// LEFT RESET SW PLS
OR        T0282	// LF_2D CODE TM OUT
OUT       M0093A	// LF_2D CODE TM OUT
; L714
LOAD      M0093B	// LF_2D CODE NG
LOAD NOT  M01700	// Mes / Mes FileZilla
AND NOT   M00008	// LEFT RESET SW PLS
LOAD      M01700	// Mes / Mes FileZilla
AND       F0009A
LOAD      M06516	// L_P&P 1st VACUUM CHECK ON
OR        P00130	// L_P&P 1st EJECT ON
AND LOAD
OR LOAD
AND LOAD
LOAD      M01810	// PLC Barcode NG Left
AND       M01700	// Mes / Mes FileZilla
OR LOAD
OR        M00358	// LF_2D CODE NG PLS
OUT       M0093B	// LF_2D CODE NG
; L719
LOAD      M0093B	// LF_2D CODE NG
AND       M01700	// Mes / Mes FileZilla
AND NOT   M06516	// L_P&P 1st VACUUM CHECK ON
AND NOT   P00130	// L_P&P 1st EJECT ON
AND       F0009A
OR        M00008	// LEFT RESET SW PLS
RST       M01810	// PLC Barcode NG Left
; L721
LOAD      M0093C	// RT_2D CODE TM OUT
AND NOT   M00008	// LEFT RESET SW PLS
OR        T0292	// RT_2D CODE TM OUT
OUT       M0093C	// RT_2D CODE TM OUT
; L723
LOAD      M0093D	// RT_2D CODE NG
LOAD NOT  M01700	// Mes / Mes FileZilla
AND NOT   M00008	// LEFT RESET SW PLS
LOAD      M01700	// Mes / Mes FileZilla
AND       F0009A
LOAD      M06616	// R_P&P 1st VACUUM CHECK ON
OR        P00160	// R_P&P 1st EJECT ON
AND LOAD
OR LOAD
AND LOAD
LOAD      M02810	// PLC Barcode NG Right
AND       M01700	// Mes / Mes FileZilla
OR LOAD
OR        M00368	// RT_2D CODE NG PLS
OUT       M0093D	// RT_2D CODE NG

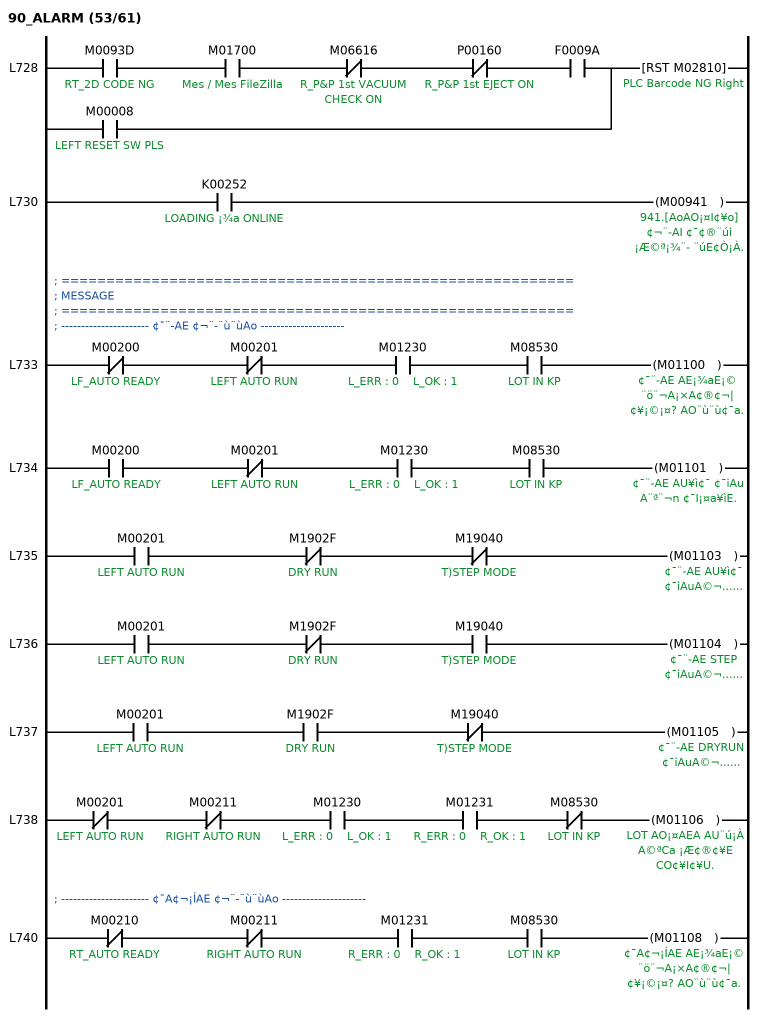
; L728
LOAD      M0093D	// RT_2D CODE NG
AND       M01700	// Mes / Mes FileZilla
AND NOT   M06616	// R_P&P 1st VACUUM CHECK ON
AND NOT   P00160	// R_P&P 1st EJECT ON
AND       F0009A
OR        M00008	// LEFT RESET SW PLS
RST       M02810	// PLC Barcode NG Right
; L730
LOAD      K00252	// LOADING ¡¾a ONLINE
OUT       M00941	// 941.[AoAO¡¤I¢¥o] ¢¬¨­AI ¢¯¢®¨úi ¡Æ©ª¡¾¨­ ¨úE¢Ò¡À.
// =========================================================
// 
//       MESSAGE
// 
// =========================================================
// ---------------------- ¢¯¨­AE ¢¬¨­¨ù¨ùAo ---------------------
; L733
LOAD NOT  M00200	// LF_AUTO READY
AND NOT   M00201	// LEFT AUTO RUN
AND       M01230	// L_ERR : 0    L_OK : 1
AND       M08530	// LOT IN KP
OUT       M01100	// ¢¯¨­AE AE¡¾aE¡© ¨ö¨¬A¡×A¢®¢¬| ¢¥¡©¡¤? AO¨ù¨ù¢¯a.
; L734
LOAD      M00200	// LF_AUTO READY
AND NOT   M00201	// LEFT AUTO RUN
AND       M01230	// L_ERR : 0    L_OK : 1
AND       M08530	// LOT IN KP
OUT       M01101	// ¢¯¨­AE AU¥ì¢¯ ¢¯iAu A¨ª¨¬n ¢¯I¡¤a¥ìE.
; L735
LOAD      M00201	// LEFT AUTO RUN
AND NOT   M1902F	// DRY RUN
AND NOT   M19040	// T)STEP MODE
OUT       M01103	// ¢¯¨­AE AU¥ì¢¯ ¢¯iAuA©¬......
; L736
LOAD      M00201	// LEFT AUTO RUN
AND NOT   M1902F	// DRY RUN
AND       M19040	// T)STEP MODE
OUT       M01104	// ¢¯¨­AE STEP ¢¯iAuA©¬......
; L737
LOAD      M00201	// LEFT AUTO RUN
AND       M1902F	// DRY RUN
AND NOT   M19040	// T)STEP MODE
OUT       M01105	// ¢¯¨­AE DRYRUN ¢¯iAuA©¬......
; L738
LOAD NOT  M00201	// LEFT AUTO RUN
AND NOT   M00211	// RIGHT AUTO RUN
AND       M01230	// L_ERR : 0    L_OK : 1
AND       M01231	// R_ERR : 0    R_OK : 1
AND NOT   M08530	// LOT IN KP
OUT       M01106	// LOT AO¡¤AEA AU¨ú¡À A©ªCa ¡Æ¢®¢¥E CO¢¥I¢¥U.
// ---------------------- ¢¯A¢¬¡ÍAE ¢¬¨­¨ù¨ùAo ---------------------
; L740
LOAD NOT  M00210	// RT_AUTO READY
AND NOT   M00211	// RIGHT AUTO RUN
AND       M01231	// R_ERR : 0    R_OK : 1
AND       M08530	// LOT IN KP
OUT       M01108	// ¢¯A¢¬¡ÍAE AE¡¾aE¡© ¨ö¨¬A¡×A¢®¢¬| ¢¥¡©¡¤? AO¨ù¨ù¢¯a.

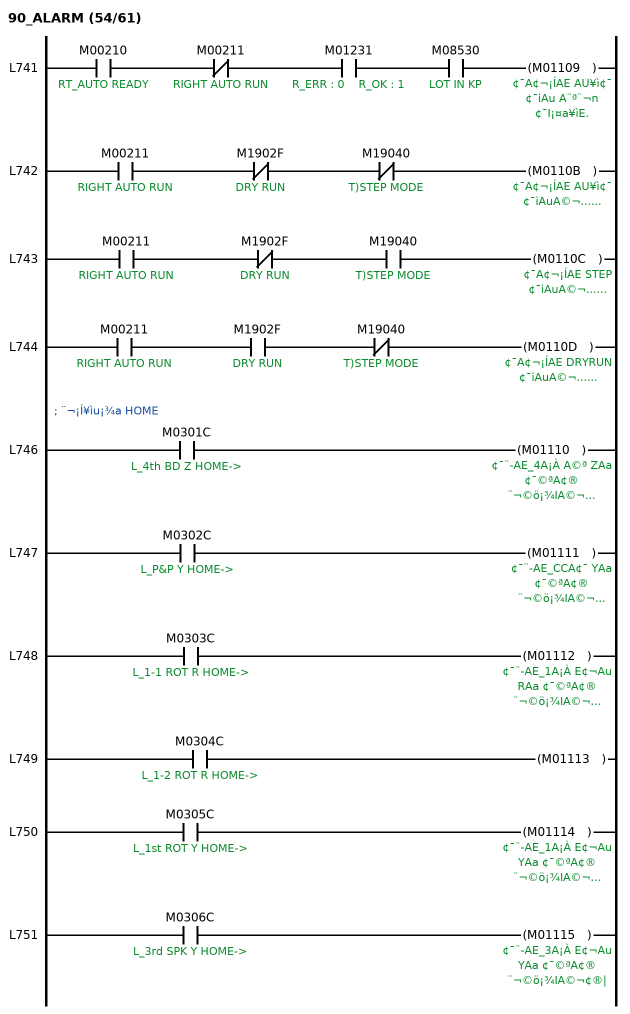
; L741
LOAD      M00210	// RT_AUTO READY
AND NOT   M00211	// RIGHT AUTO RUN
AND       M01231	// R_ERR : 0    R_OK : 1
AND       M08530	// LOT IN KP
OUT       M01109	// ¢¯A¢¬¡ÍAE AU¥ì¢¯ ¢¯iAu A¨ª¨¬n ¢¯I¡¤a¥ìE.
; L742
LOAD      M00211	// RIGHT AUTO RUN
AND NOT   M1902F	// DRY RUN
AND NOT   M19040	// T)STEP MODE
OUT       M0110B	// ¢¯A¢¬¡ÍAE AU¥ì¢¯ ¢¯iAuA©¬......
; L743
LOAD      M00211	// RIGHT AUTO RUN
AND NOT   M1902F	// DRY RUN
AND       M19040	// T)STEP MODE
OUT       M0110C	// ¢¯A¢¬¡ÍAE STEP ¢¯iAuA©¬......
; L744
LOAD      M00211	// RIGHT AUTO RUN
AND       M1902F	// DRY RUN
AND NOT   M19040	// T)STEP MODE
OUT       M0110D	// ¢¯A¢¬¡ÍAE DRYRUN ¢¯iAuA©¬......
// ¨¬¡Í¥ìu¡¾a HOME
; L746
LOAD      M0301C	// L_4th BD Z HOME->
OUT       M01110	// ¢¯¨­AE_4A¡À A©ª ZAa ¢¯©ªA¢® ¨¬©ö¡¾IA©¬...
; L747
LOAD      M0302C	// L_P&P Y HOME->
OUT       M01111	// ¢¯¨­AE_CCA¢¯ YAa ¢¯©ªA¢® ¨¬©ö¡¾IA©¬...
; L748
LOAD      M0303C	// L_1-1 ROT R HOME->
OUT       M01112	// ¢¯¨­AE_1A¡À E¢¬Au RAa ¢¯©ªA¢® ¨¬©ö¡¾IA©¬...
; L749
LOAD      M0304C	// L_1-2 ROT R HOME->
OUT       M01113
; L750
LOAD      M0305C	// L_1st ROT Y HOME->
OUT       M01114	// ¢¯¨­AE_1A¡À E¢¬Au YAa ¢¯©ªA¢® ¨¬©ö¡¾IA©¬...
; L751
LOAD      M0306C	// L_3rd SPK Y HOME->
OUT       M01115	// ¢¯¨­AE_3A¡À E¢¬Au YAa ¢¯©ªA¢® ¨¬©ö¡¾IA©¬¢®|

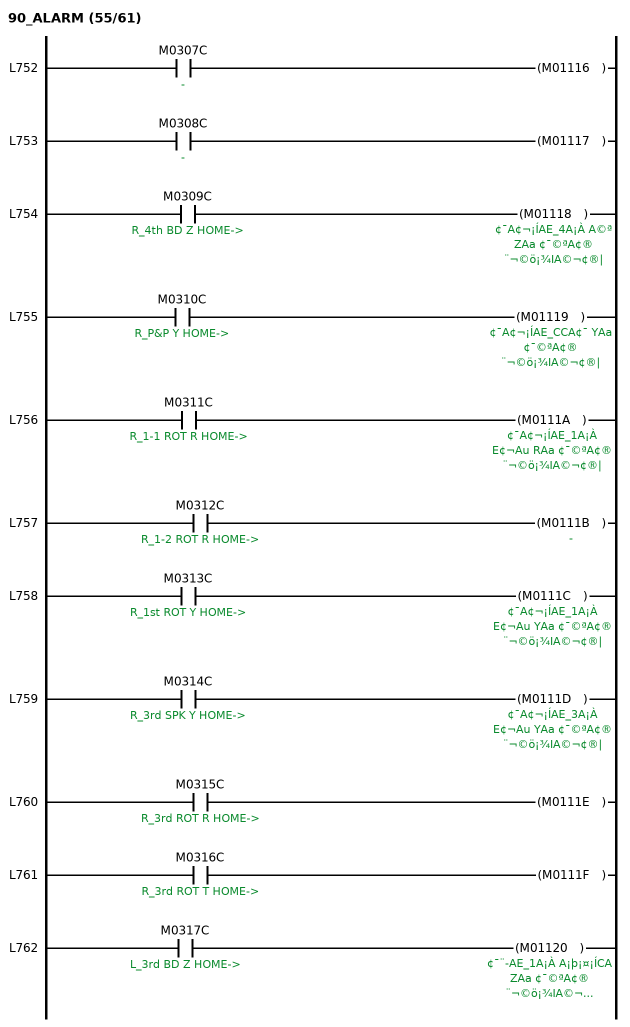
; L752
LOAD      M0307C	// -
OUT       M01116
; L753
LOAD      M0308C	// -
OUT       M01117
; L754
LOAD      M0309C	// R_4th BD Z HOME->
OUT       M01118	// ¢¯A¢¬¡ÍAE_4A¡À A©ª ZAa ¢¯©ªA¢® ¨¬©ö¡¾IA©¬¢®|
; L755
LOAD      M0310C	// R_P&P Y HOME->
OUT       M01119	// ¢¯A¢¬¡ÍAE_CCA¢¯ YAa ¢¯©ªA¢® ¨¬©ö¡¾IA©¬¢®|
; L756
LOAD      M0311C	// R_1-1 ROT R HOME->
OUT       M0111A	// ¢¯A¢¬¡ÍAE_1A¡À E¢¬Au RAa ¢¯©ªA¢® ¨¬©ö¡¾IA©¬¢®|
; L757
LOAD      M0312C	// R_1-2 ROT R HOME->
OUT       M0111B	// -
; L758
LOAD      M0313C	// R_1st ROT Y HOME->
OUT       M0111C	// ¢¯A¢¬¡ÍAE_1A¡À E¢¬Au YAa ¢¯©ªA¢® ¨¬©ö¡¾IA©¬¢®|
; L759
LOAD      M0314C	// R_3rd SPK Y HOME->
OUT       M0111D	// ¢¯A¢¬¡ÍAE_3A¡À E¢¬Au YAa ¢¯©ªA¢® ¨¬©ö¡¾IA©¬¢®|
; L760
LOAD      M0315C	// R_3rd ROT R HOME->
OUT       M0111E
; L761
LOAD      M0316C	// R_3rd ROT T HOME->
OUT       M0111F
; L762
LOAD      M0317C	// L_3rd BD Z HOME->
OUT       M01120	// ¢¯¨­AE_1A¡À A¡þ¡¤¡ÍCA ZAa ¢¯©ªA¢® ¨¬©ö¡¾IA©¬...

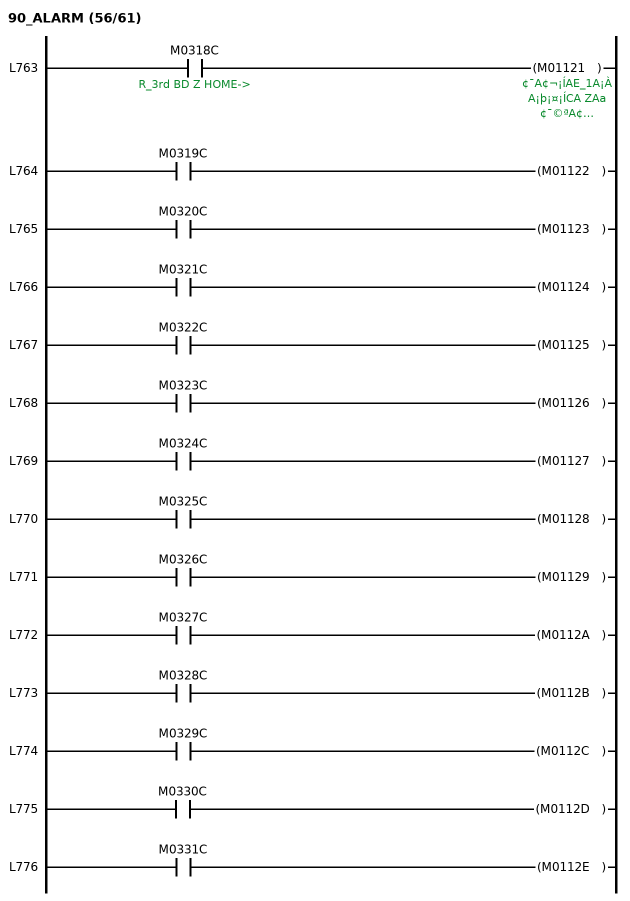
; L763
LOAD      M0318C	// R_3rd BD Z HOME->
OUT       M01121	// ¢¯A¢¬¡ÍAE_1A¡À A¡þ¡¤¡ÍCA ZAa ¢¯©ªA¢® ¨¬©ö¡¾IA©¬...
; L764
LOAD      M0319C
OUT       M01122
; L765
LOAD      M0320C
OUT       M01123
; L766
LOAD      M0321C
OUT       M01124
; L767
LOAD      M0322C
OUT       M01125
; L768
LOAD      M0323C
OUT       M01126
; L769
LOAD      M0324C
OUT       M01127
; L770
LOAD      M0325C
OUT       M01128
; L771
LOAD      M0326C
OUT       M01129
; L772
LOAD      M0327C
OUT       M0112A
; L773
LOAD      M0328C
OUT       M0112B
; L774
LOAD      M0329C
OUT       M0112C
; L775
LOAD      M0330C
OUT       M0112D
; L776
LOAD      M0331C
OUT       M0112E

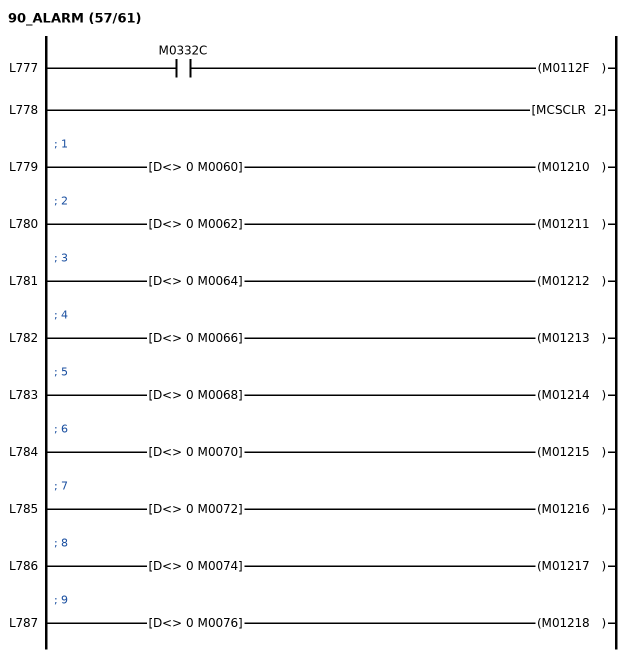
; L777
LOAD      M0332C
OUT       M0112F
; L778
MCSCLR    2
; L779
LOADD<>   0 M0060
OUT       M01210
// output comment: 1
; L780
LOADD<>   0 M0062
OUT       M01211
// output comment: 2
; L781
LOADD<>   0 M0064
OUT       M01212
// output comment: 3
; L782
LOADD<>   0 M0066
OUT       M01213
// output comment: 4
; L783
LOADD<>   0 M0068
OUT       M01214
// output comment: 5
; L784
LOADD<>   0 M0070
OUT       M01215
// output comment: 6
; L785
LOADD<>   0 M0072
OUT       M01216
// output comment: 7
; L786
LOADD<>   0 M0074
OUT       M01217
// output comment: 8
; L787
LOADD<>   0 M0076
OUT       M01218
// output comment: 9

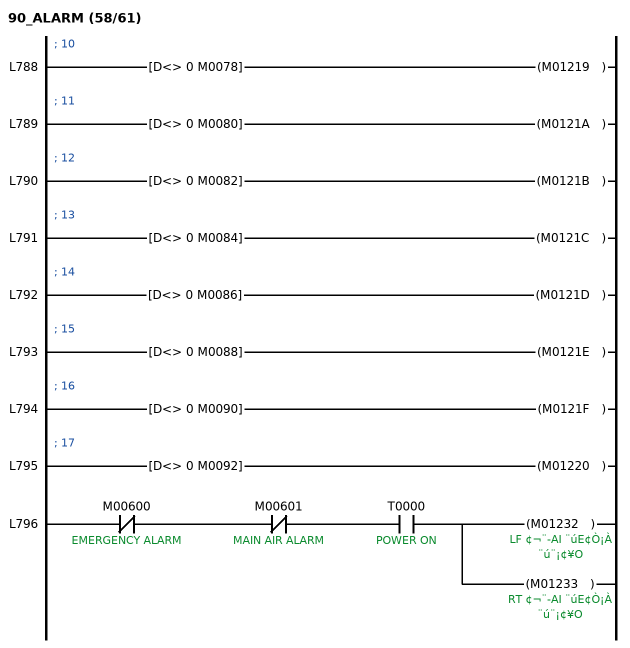
; L788
LOADD<>   0 M0078
OUT       M01219
// output comment: 10
; L789
LOADD<>   0 M0080
OUT       M0121A
// output comment: 11
; L790
LOADD<>   0 M0082
OUT       M0121B
// output comment: 12
; L791
LOADD<>   0 M0084
OUT       M0121C
// output comment: 13
; L792
LOADD<>   0 M0086
OUT       M0121D
// output comment: 14
; L793
LOADD<>   0 M0088
OUT       M0121E
// output comment: 15
; L794
LOADD<>   0 M0090
OUT       M0121F
// output comment: 16
; L795
LOADD<>   0 M0092
OUT       M01220
// output comment: 17
; L796
LOAD NOT  M00600	// EMERGENCY ALARM
AND NOT   M00601	// MAIN AIR ALARM
AND       T0000	// POWER ON
OUT       M01232	// LF ¢¬¨­AI ¨úE¢Ò¡À ¨ú¨¡¢¥O
OUT       M01233	// RT ¢¬¨­AI ¨úE¢Ò¡À ¨ú¨¡¢¥O

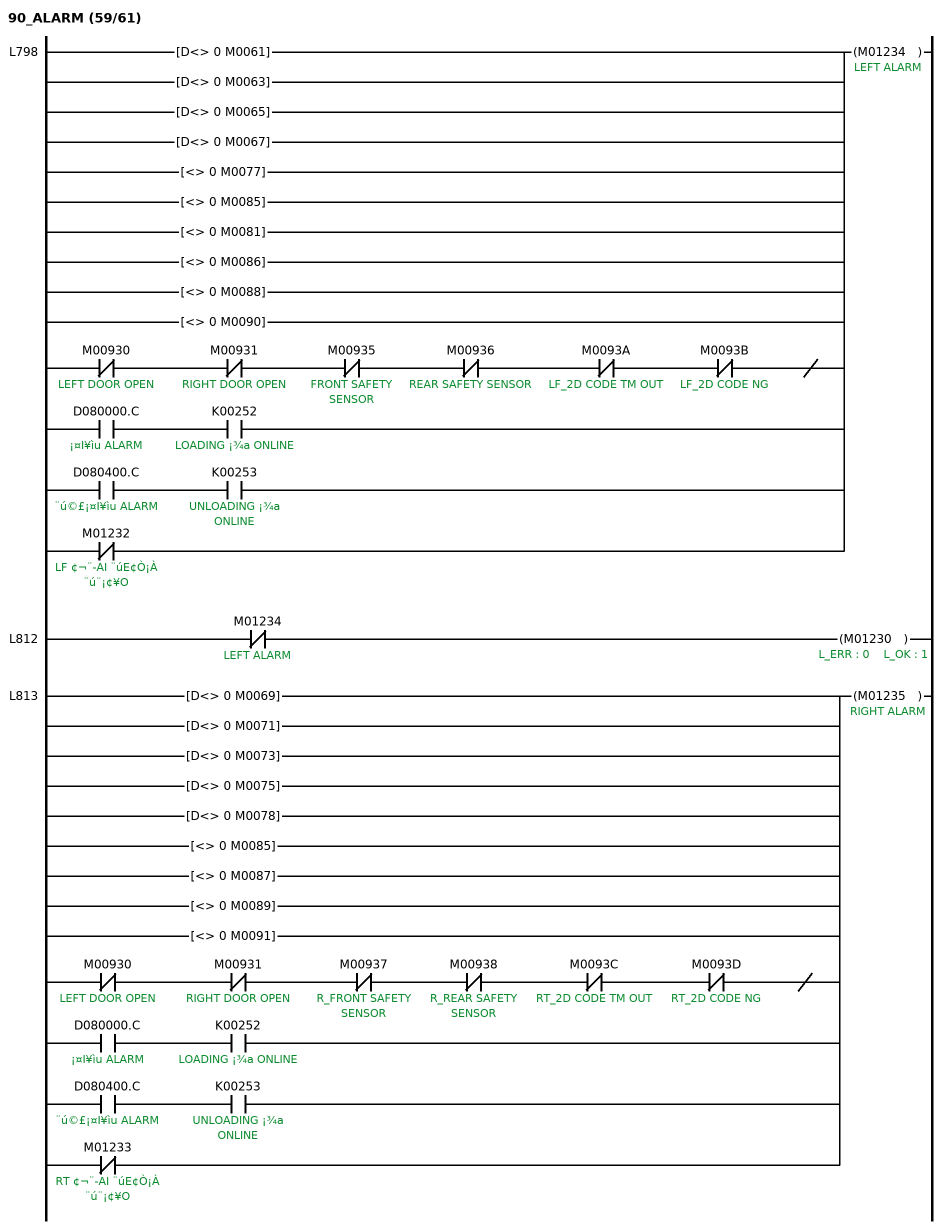
; L798
LOADD<>   0 M0061
ORD<>     0 M0063
ORD<>     0 M0065
ORD<>     0 M0067
OR<>      0 M0077
OR<>      0 M0085
OR<>      0 M0081
OR<>      0 M0086
OR<>      0 M0088
OR<>      0 M0090
LOAD NOT  M00930	// LEFT DOOR OPEN
AND NOT   M00931	// RIGHT DOOR OPEN
AND NOT   M00935	// FRONT SAFETY SENSOR
AND NOT   M00936	// REAR SAFETY SENSOR
AND NOT   M0093A	// LF_2D CODE TM OUT
AND NOT   M0093B	// LF_2D CODE NG
NOT
OR LOAD
LOAD      D080000.C	// ¡¤I¥ìu ALARM
AND       K00252	// LOADING ¡¾a ONLINE
OR LOAD
LOAD      D080400.C	// ¨ú©£¡¤I¥ìu ALARM
AND       K00253	// UNLOADING ¡¾a ONLINE
OR LOAD
OR NOT    M01232	// LF ¢¬¨­AI ¨úE¢Ò¡À ¨ú¨¡¢¥O
OUT       M01234	// LEFT ALARM
; L812
LOAD NOT  M01234	// LEFT ALARM
OUT       M01230	// L_ERR : 0    L_OK : 1
; L813
LOADD<>   0 M0069
ORD<>     0 M0071
ORD<>     0 M0073
ORD<>     0 M0075
ORD<>     0 M0078
OR<>      0 M0085
OR<>      0 M0087
OR<>      0 M0089
OR<>      0 M0091
LOAD NOT  M00930	// LEFT DOOR OPEN
AND NOT   M00931	// RIGHT DOOR OPEN
AND NOT   M00937	// R_FRONT SAFETY SENSOR
AND NOT   M00938	// R_REAR SAFETY SENSOR
AND NOT   M0093C	// RT_2D CODE TM OUT
AND NOT   M0093D	// RT_2D CODE NG
NOT
OR LOAD
LOAD      D080000.C	// ¡¤I¥ìu ALARM
AND       K00252	// LOADING ¡¾a ONLINE
OR LOAD
LOAD      D080400.C	// ¨ú©£¡¤I¥ìu ALARM
AND       K00253	// UNLOADING ¡¾a ONLINE
OR LOAD
OR NOT    M01233	// RT ¢¬¨­AI ¨úE¢Ò¡À ¨ú¨¡¢¥O
OUT       M01235	// RIGHT ALARM

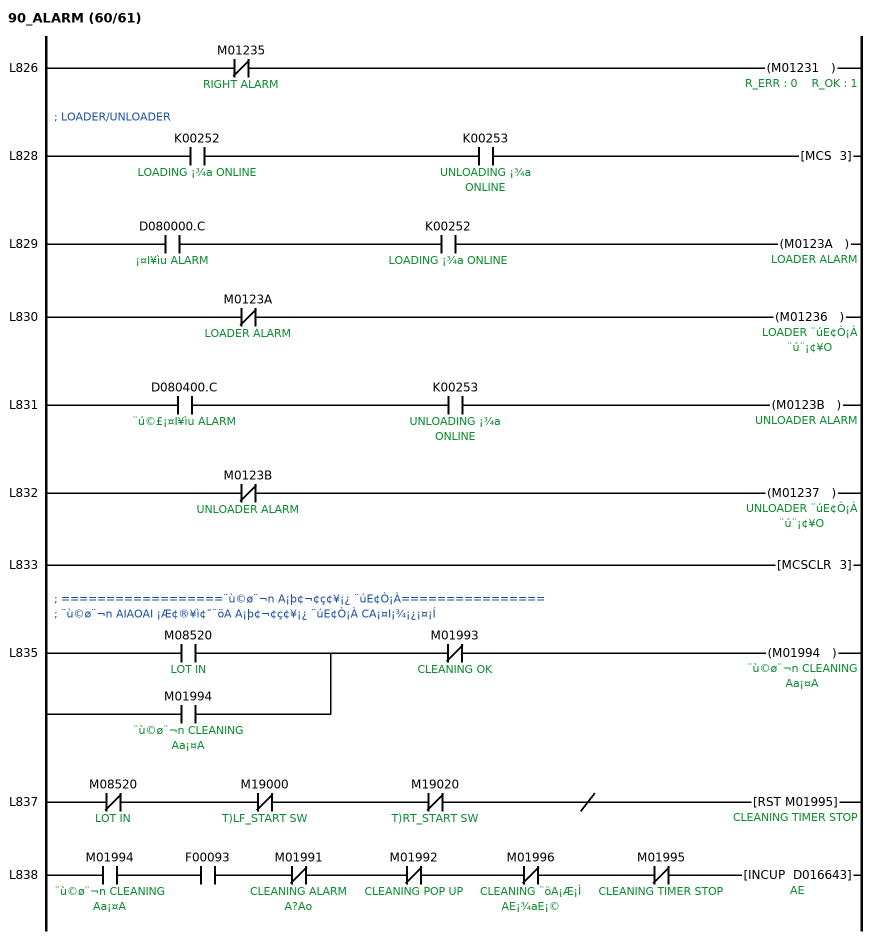
; L826
LOAD NOT  M01235	// RIGHT ALARM
OUT       M01231	// R_ERR : 0    R_OK : 1
// LOADER/UNLOADER
; L828
LOAD      K00252	// LOADING ¡¾a ONLINE
AND       K00253	// UNLOADING ¡¾a ONLINE
MCS       3
; L829
LOAD      D080000.C	// ¡¤I¥ìu ALARM
AND       K00252	// LOADING ¡¾a ONLINE
OUT       M0123A	// LOADER ALARM
; L830
LOAD NOT  M0123A	// LOADER ALARM
OUT       M01236	// LOADER ¨úE¢Ò¡À ¨ú¨¡¢¥O
; L831
LOAD      D080400.C	// ¨ú©£¡¤I¥ìu ALARM
AND       K00253	// UNLOADING ¡¾a ONLINE
OUT       M0123B	// UNLOADER ALARM
; L832
LOAD NOT  M0123B	// UNLOADER ALARM
OUT       M01237	// UNLOADER ¨úE¢Ò¡À ¨ú¨¡¢¥O
; L833
MCSCLR    3
// ==================¨ù©ø¨¬n A¡þ¢¬¢ç¢¥¡¿ ¨úE¢Ò¡À================
; L835
LOAD      M08520	// LOT IN
OR        M01994	// ¨ù©ø¨¬n CLEANING Aa¡¤A
AND NOT   M01993	// CLEANING OK
OUT       M01994	// ¨ù©ø¨¬n CLEANING Aa¡¤A
// output comment: ¨ù©ø¨¬n AIAOAI ¡Æ¢®¥ì¢¯¨öA A¡þ¢¬¢ç¢¥¡¿ ¨úE¢Ò¡À CA¡¤I¡¾¡¿¡¤¡Í
; L837
LOAD NOT  M08520	// LOT IN
AND NOT   M19000	// T)LF_START SW
AND NOT   M19020	// T)RT_START SW
NOT
RST       M01995	// CLEANING TIMER STOP
; L838
LOAD      M01994	// ¨ù©ø¨¬n CLEANING Aa¡¤A
AND       F00093
AND NOT   M01991	// CLEANING ALARM A?Ao
AND NOT   M01992	// CLEANING POP UP
AND NOT   M01996	// CLEANING ¨öA¡Æ¡Ì AE¡¾aE¡©
AND NOT   M01995	// CLEANING TIMER STOP
INCUP     D016643	// AE

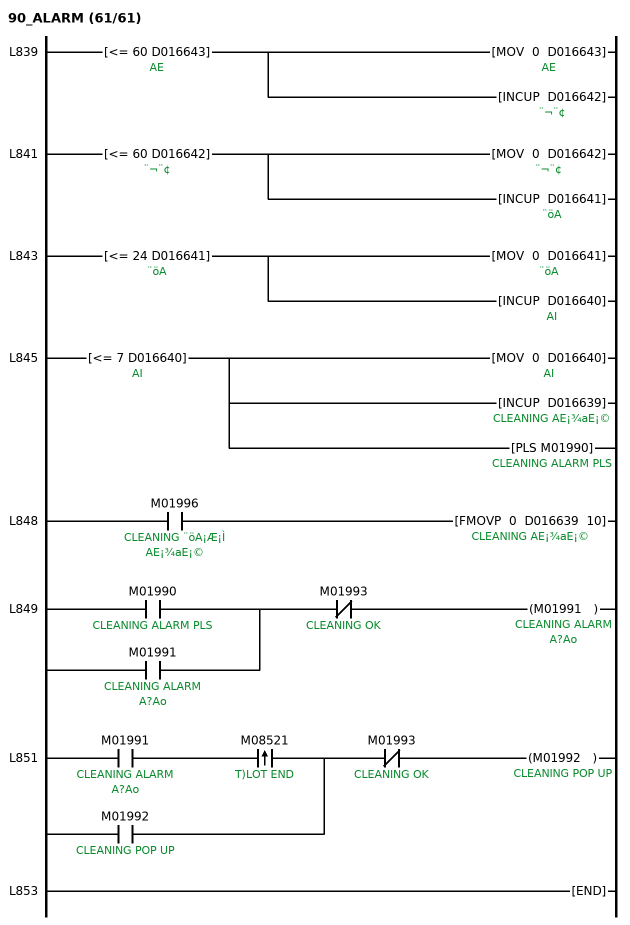
; L839
LOAD<=    60 D016643	// AE
MOV       0 D016643	// AE
INCUP     D016642	// ¨¬¨¢
; L841
LOAD<=    60 D016642	// ¨¬¨¢
MOV       0 D016642	// ¨¬¨¢
INCUP     D016641	// ¨öA
; L843
LOAD<=    24 D016641	// ¨öA
MOV       0 D016641	// ¨öA
INCUP     D016640	// AI
; L845
LOAD<=    7 D016640	// AI
MOV       0 D016640	// AI
INCUP     D016639	// CLEANING AE¡¾aE¡©
OUTP      M01990	// CLEANING ALARM PLS
; L848
LOAD      M01996	// CLEANING ¨öA¡Æ¡Ì AE¡¾aE¡©
FMOVP     0 D016639 10	// CLEANING AE¡¾aE¡©
; L849
LOAD      M01990	// CLEANING ALARM PLS
OR        M01991	// CLEANING ALARM A?Ao
AND NOT   M01993	// CLEANING OK
OUT       M01991	// CLEANING ALARM A?Ao
; L851
LOAD      M01991	// CLEANING ALARM A?Ao
ANDP      M08521	// T)LOT END
OR        M01992	// CLEANING POP UP
AND NOT   M01993	// CLEANING OK
OUT       M01992	// CLEANING POP UP
; L853
END

PROGRAM 91_DEVICE_CHANGE (task: ¨ö¨¬A¥ì CA¡¤I¡¾¡¿¡¤¡Í)

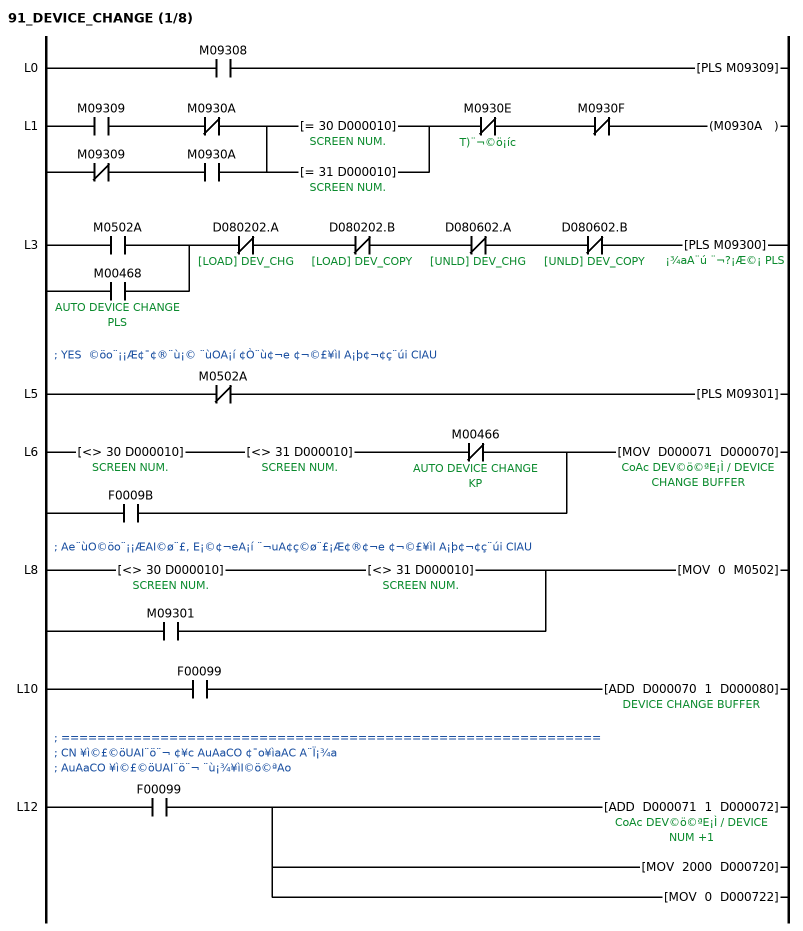
; L0
LOAD      M09308
OUTP      M09309
; L1
LOAD      M09309
AND NOT   M0930A
LOAD NOT  M09309
AND       M0930A
OR LOAD
LOAD=     30 D000010	// SCREEN NUM.
OR=       31 D000010	// SCREEN NUM.
AND LOAD
AND NOT   M0930E	// T)¨¬©ö¡íc
AND NOT   M0930F
OUT       M0930A
; L3
LOAD      M0502A
OR        M00468	// AUTO DEVICE CHANGE PLS
AND NOT   D080202.A	// [LOAD] DEV_CHG
AND NOT   D080202.B	// [LOAD] DEV_COPY
AND NOT   D080602.A	// [UNLD] DEV_CHG
AND NOT   D080602.B	// [UNLD] DEV_COPY
OUTP      M09300	// ¡¾aA¨ú ¨¬?¡Æ©¡ PLS
; L5
LOAD NOT  M0502A
OUTP      M09301
// output comment: YES  ©öo¨¡¡Æ¢¯¢®¨ù¡© ¨ùOA¡í ¢Ò¨ù¢¬e ¢¬©£¥ìI A¡þ¢¬¢ç¨úi CIAU
; L6
LOAD<>    30 D000010	// SCREEN NUM.
AND<>     31 D000010	// SCREEN NUM.
AND NOT   M00466	// AUTO DEVICE CHANGE KP
OR        F0009B
MOV       D000071 D000070	// CoAc DEV©ö©ªE¡Ì / DEVICE CHANGE BUFFER
; L8
LOAD<>    30 D000010	// SCREEN NUM.
AND<>     31 D000010	// SCREEN NUM.
OR        M09301
MOV       0 M0502
// output comment: Ae¨ùO©öo¨¡¡ÆAI©ø¨£, E¡©¢¬eA¡í ¨¬uA¢ç©ø¨£¡Æ¢®¢¬e ¢¬©£¥ìI A¡þ¢¬¢ç¨úi CIAU
; L10
LOAD      F00099
ADD       D000070 1 D000080	// DEVICE CHANGE BUFFER
// ============================================================
; L12
LOAD      F00099
ADD       D000071 1 D000072	// CoAc DEV©ö©ªE¡Ì / DEVICE NUM +1
MOV       2000 D000720
MOV       0 D000722
// output comment: CN ¥ì©£©öUAI¨ö¨¬ ¢¥c AuAaCO ¢¯o¥ìaAC A¨Ï¡¾a
// output comment: AuAaCO ¥ì©£©öUAI¨ö¨¬ ¨ù¡¾¥ìI©ö©ªAo

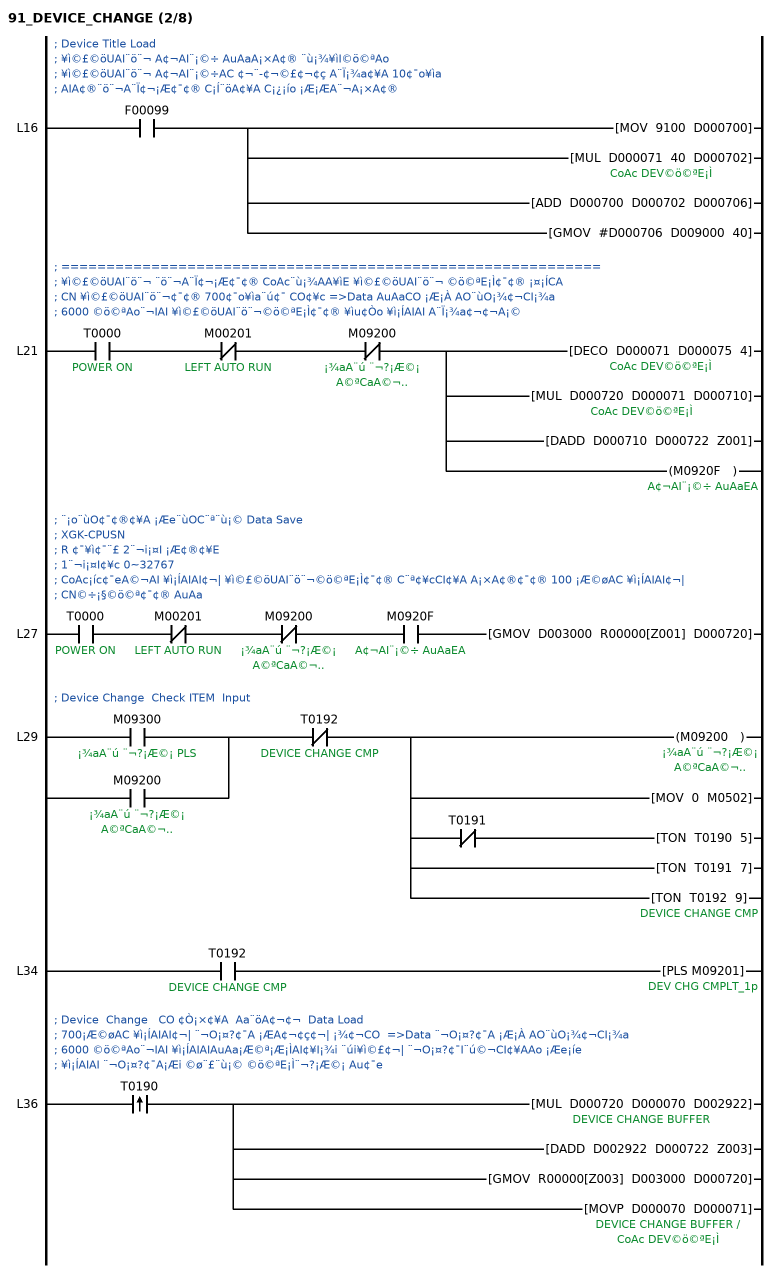
// Device Title Load
; L16
LOAD      F00099
MOV       9100 D000700
MUL       D000071 40 D000702	// CoAc DEV©ö©ªE¡Ì
ADD       D000700 D000702 D000706
GMOV      #D000706 D009000 40
// output comment: ¥ì©£©öUAI¨ö¨¬ A¢¬AI¨¡©÷ AuAaA¡×A¢® ¨ù¡¾¥ìI©ö©ªAo
// output comment: ¥ì©£©öUAI¨ö¨¬ A¢¬AI¨¡©÷AC ¢¬¨­¢¬©£¢¬¢ç A¨Ï¡¾a¢¥A 10¢¯o¥ìa
// output comment: AIA¢®¨ö¨¬A¨Ï¢¬¡Æ¢¯¢® C¡Í¨öA¢¥A C¡¿¡ío ¡Æ¡ÆA¨¬A¡×A¢®
// ============================================================
; L21
LOAD      T0000	// POWER ON
AND NOT   M00201	// LEFT AUTO RUN
AND NOT   M09200	// ¡¾aA¨ú ¨¬?¡Æ©¡ A©ªCaA©¬..
DECO      D000071 D000075 4	// CoAc DEV©ö©ªE¡Ì
MUL       D000720 D000071 D000710	// CoAc DEV©ö©ªE¡Ì
DADD      D000710 D000722 Z001
OUT       M0920F	// A¢¬AI¨¡©÷ AuAaEA
// output comment: ¥ì©£©öUAI¨ö¨¬ ¨ö¨¬A¨Ï¢¬¡Æ¢¯¢® CoAc¨ù¡¾AA¥ìE ¥ì©£©öUAI¨ö¨¬ ©ö©ªE¡Ì¢¯¢® ¡¤¡ÍCA
// output comment: CN ¥ì©£©öUAI¨ö¨¬¢¯¢® 700¢¯o¥ìa¨ú¢¯ CO¢¥c =>Data AuAaCO ¡Æ¡À AO¨ùO¡¾¢¬CI¡¾a
// output comment: 6000 ©ö©ªAo¨¬IAI ¥ì©£©öUAI¨ö¨¬©ö©ªE¡Ì¢¯¢® ¥ìu¢Òo ¥ì¡ÍAIAI A¨Ï¡¾a¢¬¢¬A¡©
// ¨¡o¨ùO¢¯¢®¢¥A ¡Æe¨ùOC¨ª¨ù¡© Data Save
// XGK-CPUSN
// R ¢¯¥ì¢¯¨£ 2¨¬i¡¤I ¡Æ¢®¢¥E
// 1¨¬i¡¤I¢¥c 0~32767
; L27
LOAD      T0000	// POWER ON
AND NOT   M00201	// LEFT AUTO RUN
AND NOT   M09200	// ¡¾aA¨ú ¨¬?¡Æ©¡ A©ªCaA©¬..
AND       M0920F	// A¢¬AI¨¡©÷ AuAaEA
GMOV      D003000 R00000[Z001] D000720
// output comment: CoAc¡íc¢¯eA©¬AI ¥ì¡ÍAIAI¢¬| ¥ì©£©öUAI¨ö¨¬©ö©ªE¡Ì¢¯¢® C¨ª¢¥cCI¢¥A A¡×A¢®¢¯¢® 100 ¡Æ©øAC ¥ì¡ÍAIAI¢¬| CN©÷¡§©ö©ª¢¯¢® AuAa
// Device Change  Check ITEM  Input
; L29
LOAD      M09300	// ¡¾aA¨ú ¨¬?¡Æ©¡ PLS
OR        M09200	// ¡¾aA¨ú ¨¬?¡Æ©¡ A©ªCaA©¬..
AND NOT   T0192	// DEVICE CHANGE CMP
OUT       M09200	// ¡¾aA¨ú ¨¬?¡Æ©¡ A©ªCaA©¬..
MOV       0 M0502
MPUSH
AND NOT   T0191
TON       T0190 5
MPOP
TON       T0191 7
TON       T0192 9	// DEVICE CHANGE CMP
; L34
LOAD      T0192	// DEVICE CHANGE CMP
OUTP      M09201	// DEV CHG CMPLT_1p
// Device  Change   CO ¢Ò¡×¢¥A  Aa¨öA¢¬¢¬  Data Load
; L36
LOADP     T0190
MUL       D000720 D000070 D002922	// DEVICE CHANGE BUFFER
DADD      D002922 D000722 Z003
GMOV      R00000[Z003] D003000 D000720
MOVP      D000070 D000071	// DEVICE CHANGE BUFFER / CoAc DEV©ö©ªE¡Ì
// output comment: 700¡Æ©øAC ¥ì¡ÍAIAI¢¬| ¨¬O¡¤?¢¯A ¡ÆA¢¬¢ç¢¬| ¡¾¢¬CO  =>Data ¨¬O¡¤?¢¯A ¡Æ¡À AO¨ùO¡¾¢¬CI¡¾a
// output comment: 6000 ©ö©ªAo¨¬IAI ¥ì¡ÍAIAIAuAa¡Æ©ª¡Æ¡ÌAI¢¥I¡¾i ¨úi¥ì©£¢¬| ¨¬O¡¤?¢¯I¨ú©¬CI¢¥AAo ¡Æe¡íe
// output comment: ¥ì¡ÍAIAI ¨¬O¡¤?¢¯A¡Æi ©ø¨£¨ù¡© ©ö©ªE¡Ì¨¬?¡Æ©¡ Au¢¯e

